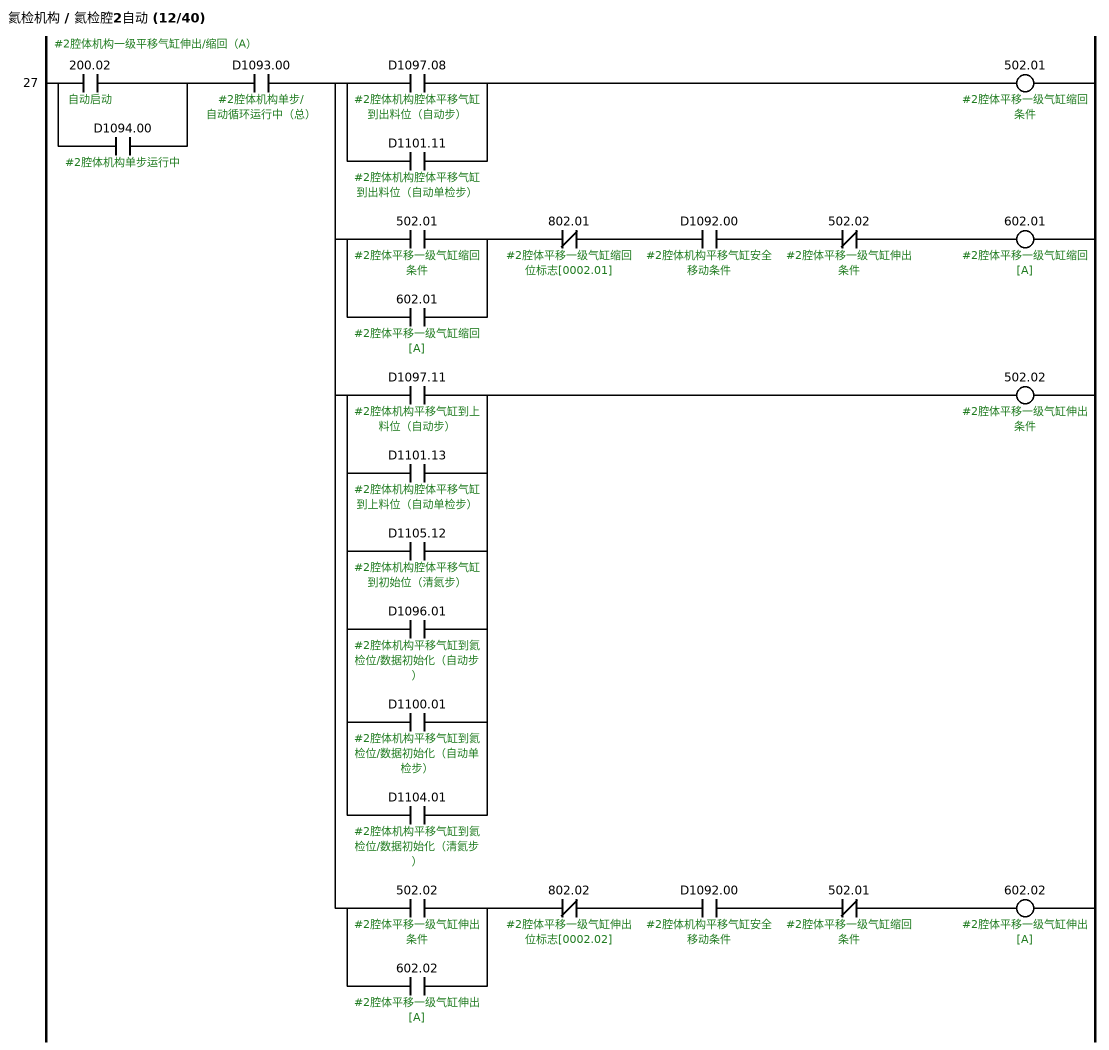
; [picture p264: 氦检机构 / 氦检腔2自动, rungs 27-27]
; rung 27: #2腔体机构一级平移气缸伸出/缩回（A）
LD 200.02  ; 自动启动
OR D1094.00  ; #2腔体机构单步运行中
AND D1093.00  ; #2腔体机构单步/自动循环运行中（总）
OUT TR0
LD D1097.08  ; #2腔体机构腔体平移气缸到出料位（自动步）
OR D1101.11  ; #2腔体机构腔体平移气缸到出料位（自动单检步）
ANDLD
OUT 502.01  ; #2腔体平移一级气缸缩回条件
LD TR0
LD 502.01  ; #2腔体平移一级气缸缩回条件
OR 602.01  ; #2腔体平移一级气缸缩回[A]
ANDLD
ANDNOT 802.01  ; #2腔体平移一级气缸缩回位标志[0002.01]
AND D1092.00  ; #2腔体机构平移气缸安全移动条件
ANDNOT 502.02  ; #2腔体平移一级气缸伸出条件
OUT 602.01  ; #2腔体平移一级气缸缩回[A]
LD TR0
LD D1097.11  ; #2腔体机构平移气缸到上料位（自动步）
OR D1101.13  ; #2腔体机构腔体平移气缸到上料位（自动单检步）
OR D1105.12  ; #2腔体机构腔体平移气缸到初始位（清氦步）
OR D1096.01  ; #2腔体机构平移气缸到氦检位/数据初始化（自动步）
OR D1100.01  ; #2腔体机构平移气缸到氦检位/数据初始化（自动单检步）
OR D1104.01  ; #2腔体机构平移气缸到氦检位/数据初始化（清氦步）
ANDLD
OUT 502.02  ; #2腔体平移一级气缸伸出条件
LD TR0
LD 502.02  ; #2腔体平移一级气缸伸出条件
OR 602.02  ; #2腔体平移一级气缸伸出[A]
ANDLD
ANDNOT 802.02  ; #2腔体平移一级气缸伸出位标志[0002.02]
AND D1092.00  ; #2腔体机构平移气缸安全移动条件
ANDNOT 502.01  ; #2腔体平移一级气缸缩回条件
OUT 602.02  ; #2腔体平移一级气缸伸出[A]

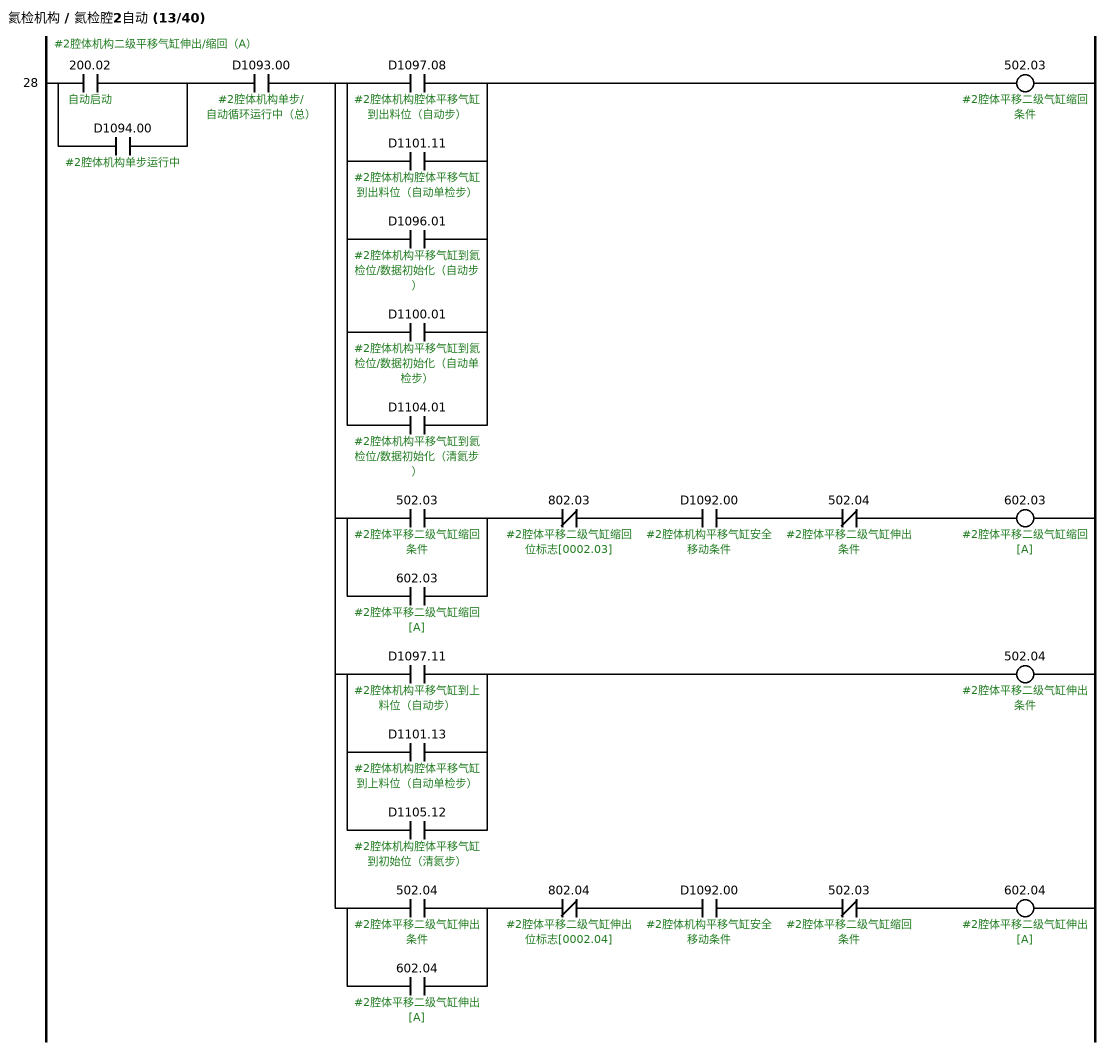
; rung 28: #2腔体机构二级平移气缸伸出/缩回（A）
LD 200.02  ; 自动启动
OR D1094.00  ; #2腔体机构单步运行中
AND D1093.00  ; #2腔体机构单步/自动循环运行中（总）
OUT TR0
LD D1097.08  ; #2腔体机构腔体平移气缸到出料位（自动步）
OR D1101.11  ; #2腔体机构腔体平移气缸到出料位（自动单检步）
OR D1096.01  ; #2腔体机构平移气缸到氦检位/数据初始化（自动步）
OR D1100.01  ; #2腔体机构平移气缸到氦检位/数据初始化（自动单检步）
OR D1104.01  ; #2腔体机构平移气缸到氦检位/数据初始化（清氦步）
ANDLD
OUT 502.03  ; #2腔体平移二级气缸缩回条件
LD TR0
LD 502.03  ; #2腔体平移二级气缸缩回条件
OR 602.03  ; #2腔体平移二级气缸缩回[A]
ANDLD
ANDNOT 802.03  ; #2腔体平移二级气缸缩回位标志[0002.03]
AND D1092.00  ; #2腔体机构平移气缸安全移动条件
ANDNOT 502.04  ; #2腔体平移二级气缸伸出条件
OUT 602.03  ; #2腔体平移二级气缸缩回[A]
LD TR0
LD D1097.11  ; #2腔体机构平移气缸到上料位（自动步）
OR D1101.13  ; #2腔体机构腔体平移气缸到上料位（自动单检步）
OR D1105.12  ; #2腔体机构腔体平移气缸到初始位（清氦步）
ANDLD
OUT 502.04  ; #2腔体平移二级气缸伸出条件
LD TR0
LD 502.04  ; #2腔体平移二级气缸伸出条件
OR 602.04  ; #2腔体平移二级气缸伸出[A]
ANDLD
ANDNOT 802.04  ; #2腔体平移二级气缸伸出位标志[0002.04]
AND D1092.00  ; #2腔体机构平移气缸安全移动条件
ANDNOT 502.03  ; #2腔体平移二级气缸缩回条件
OUT 602.04  ; #2腔体平移二级气缸伸出[A]

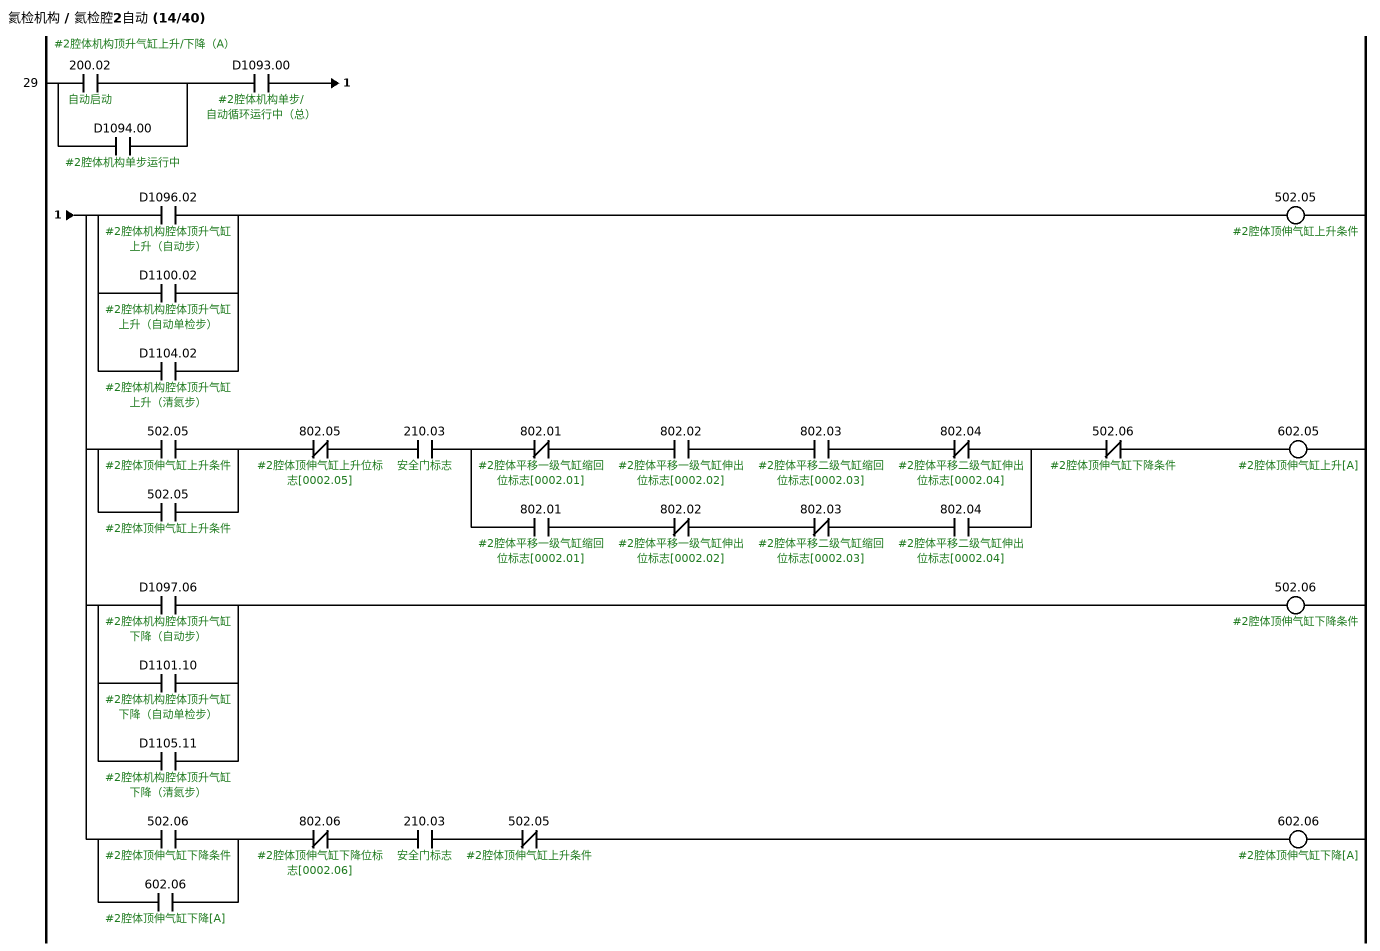
; rung 29: #2腔体机构顶升气缸上升/下降（A）
LD 200.02  ; 自动启动
OR D1094.00  ; #2腔体机构单步运行中
AND D1093.00  ; #2腔体机构单步/自动循环运行中（总）
OUT TR0
LD D1096.02  ; #2腔体机构腔体顶升气缸上升（自动步）
OR D1100.02  ; #2腔体机构腔体顶升气缸上升（自动单检步）
OR D1104.02  ; #2腔体机构腔体顶升气缸上升（清氦步）
ANDLD
OUT 502.05  ; #2腔体顶伸气缸上升条件
LD TR0
LD 502.05  ; #2腔体顶伸气缸上升条件
OR 502.05  ; #2腔体顶伸气缸上升条件
ANDLD
ANDNOT 802.05  ; #2腔体顶伸气缸上升位标志[0002.05]
AND 210.03  ; 安全门标志
LDNOT 802.01  ; #2腔体平移一级气缸缩回位标志[0002.01]
AND 802.02  ; #2腔体平移一级气缸伸出位标志[0002.02]
AND 802.03  ; #2腔体平移二级气缸缩回位标志[0002.03]
ANDNOT 802.04  ; #2腔体平移二级气缸伸出位标志[0002.04]
LD 802.01  ; #2腔体平移一级气缸缩回位标志[0002.01]
ANDNOT 802.02  ; #2腔体平移一级气缸伸出位标志[0002.02]
ANDNOT 802.03  ; #2腔体平移二级气缸缩回位标志[0002.03]
AND 802.04  ; #2腔体平移二级气缸伸出位标志[0002.04]
ORLD
ANDLD
ANDNOT 502.06  ; #2腔体顶伸气缸下降条件
OUT 602.05  ; #2腔体顶伸气缸上升[A]
LD TR0
LD D1097.06  ; #2腔体机构腔体顶升气缸下降（自动步）
OR D1101.10  ; #2腔体机构腔体顶升气缸下降（自动单检步）
OR D1105.11  ; #2腔体机构腔体顶升气缸下降（清氦步）
ANDLD
OUT 502.06  ; #2腔体顶伸气缸下降条件
LD TR0
LD 502.06  ; #2腔体顶伸气缸下降条件
OR 602.06  ; #2腔体顶伸气缸下降[A]
ANDLD
ANDNOT 802.06  ; #2腔体顶伸气缸下降位标志[0002.06]
AND 210.03  ; 安全门标志
ANDNOT 502.05  ; #2腔体顶伸气缸上升条件
OUT 602.06  ; #2腔体顶伸气缸下降[A]

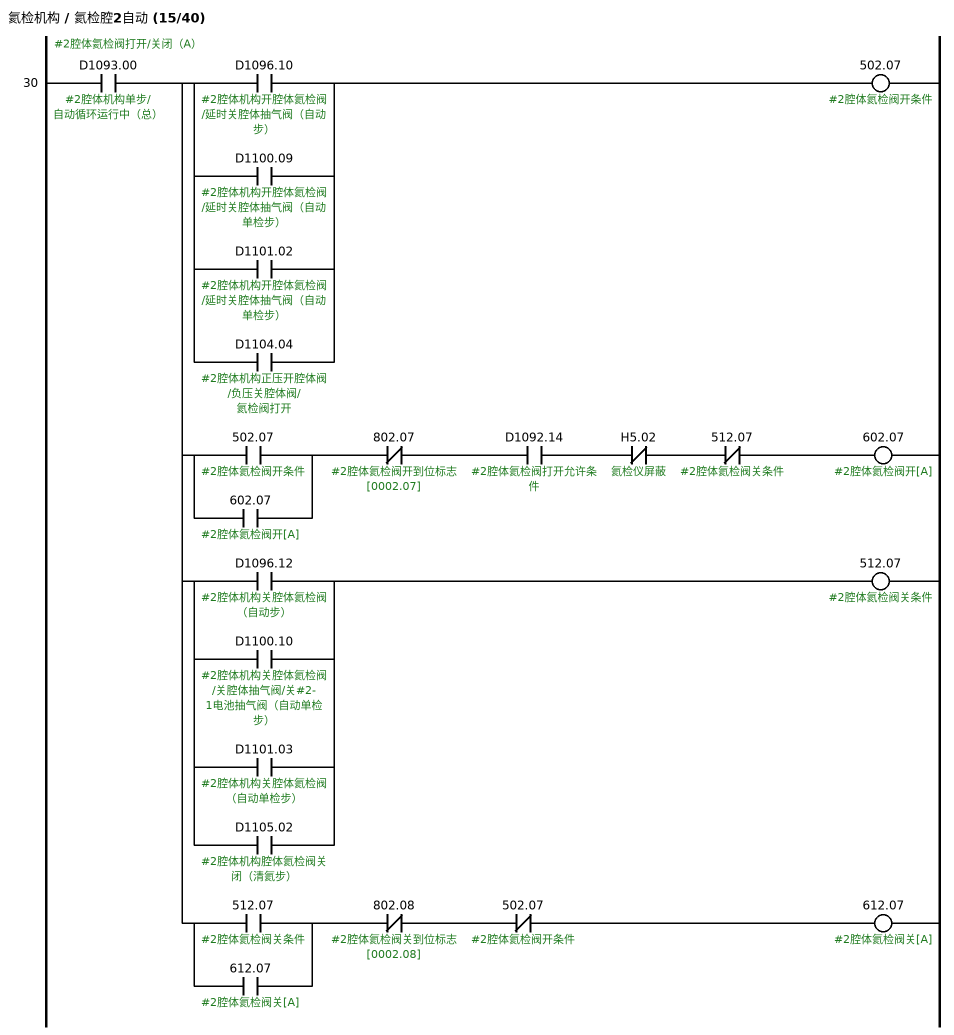
; rung 30: #2腔体氦检阀打开/关闭（A）
LD D1093.00  ; #2腔体机构单步/自动循环运行中（总）
OUT TR0
LD D1096.10  ; #2腔体机构开腔体氦检阀/延时关腔体抽气阀（自动步）
OR D1100.09  ; #2腔体机构开腔体氦检阀/延时关腔体抽气阀（自动单检步）
OR D1101.02  ; #2腔体机构开腔体氦检阀/延时关腔体抽气阀（自动单检步）
OR D1104.04  ; #2腔体机构正压开腔体阀/负压关腔体阀/氦检阀打开
ANDLD
OUT 502.07  ; #2腔体氦检阀开条件
LD TR0
LD 502.07  ; #2腔体氦检阀开条件
OR 602.07  ; #2腔体氦检阀开[A]
ANDLD
ANDNOT 802.07  ; #2腔体氦检阀开到位标志[0002.07]
AND D1092.14  ; #2腔体氦检阀打开允许条件
ANDNOT H5.02  ; 氦检仪屏蔽
ANDNOT 512.07  ; #2腔体氦检阀关条件
OUT 602.07  ; #2腔体氦检阀开[A]
LD TR0
LD D1096.12  ; #2腔体机构关腔体氦检阀（自动步）
OR D1100.10  ; #2腔体机构关腔体氦检阀/关腔体抽气阀/关#2-1电池抽气阀（自动单检步）
OR D1101.03  ; #2腔体机构关腔体氦检阀（自动单检步）
OR D1105.02  ; #2腔体机构腔体氦检阀关闭（清氦步）
ANDLD
OUT 512.07  ; #2腔体氦检阀关条件
LD TR0
LD 512.07  ; #2腔体氦检阀关条件
OR 612.07  ; #2腔体氦检阀关[A]
ANDLD
ANDNOT 802.08  ; #2腔体氦检阀关到位标志[0002.08]
ANDNOT 502.07  ; #2腔体氦检阀开条件
OUT 612.07  ; #2腔体氦检阀关[A]

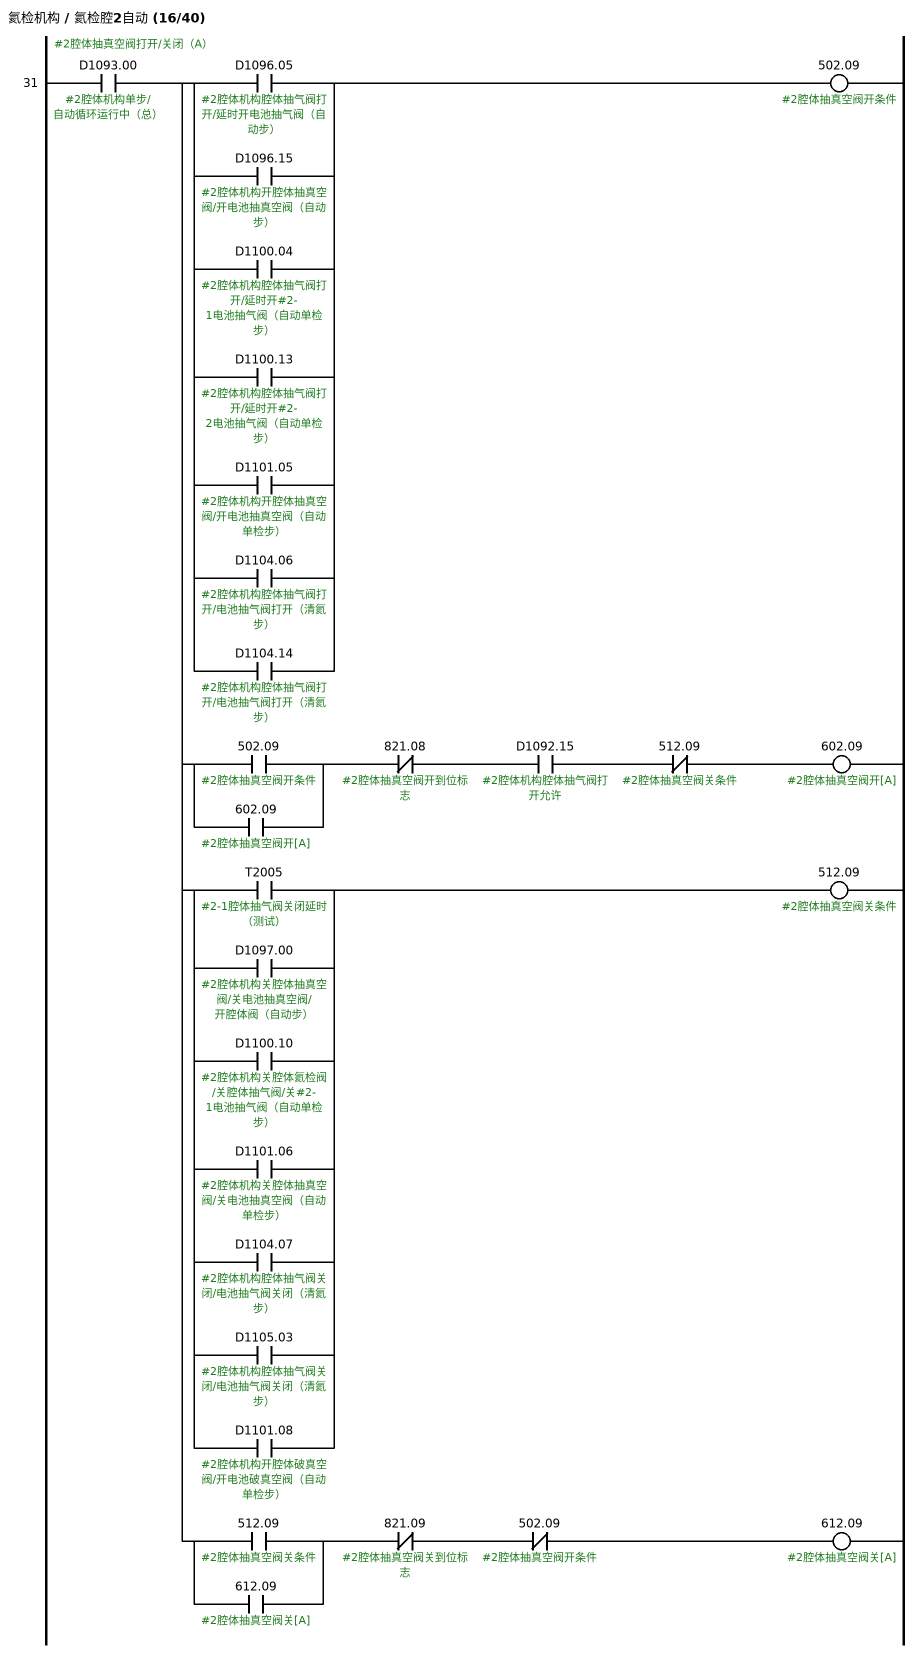
; rung 31: #2腔体抽真空阀打开/关闭（A）
LD D1093.00  ; #2腔体机构单步/自动循环运行中（总）
OUT TR0
LD D1096.05  ; #2腔体机构腔体抽气阀打开/延时开电池抽气阀（自动步）
OR D1096.15  ; #2腔体机构开腔体抽真空阀/开电池抽真空阀（自动步）
OR D1100.04  ; #2腔体机构腔体抽气阀打开/延时开#2-1电池抽气阀（自动单检步）
OR D1100.13  ; #2腔体机构腔体抽气阀打开/延时开#2-2电池抽气阀（自动单检步）
OR D1101.05  ; #2腔体机构开腔体抽真空阀/开电池抽真空阀（自动单检步）
OR D1104.06  ; #2腔体机构腔体抽气阀打开/电池抽气阀打开（清氦步）
OR D1104.14  ; #2腔体机构腔体抽气阀打开/电池抽气阀打开（清氦步）
ANDLD
OUT 502.09  ; #2腔体抽真空阀开条件
LD TR0
LD 502.09  ; #2腔体抽真空阀开条件
OR 602.09  ; #2腔体抽真空阀开[A]
ANDLD
ANDNOT 821.08  ; #2腔体抽真空阀开到位标志
AND D1092.15  ; #2腔体机构腔体抽气阀打开允许
ANDNOT 512.09  ; #2腔体抽真空阀关条件
OUT 602.09  ; #2腔体抽真空阀开[A]
LD TR0
LD T2005  ; #2-1腔体抽气阀关闭延时（测试）
OR D1097.00  ; #2腔体机构关腔体抽真空阀/关电池抽真空阀/开腔体阀（自动步）
OR D1100.10  ; #2腔体机构关腔体氦检阀/关腔体抽气阀/关#2-1电池抽气阀（自动单检步）
OR D1101.06  ; #2腔体机构关腔体抽真空阀/关电池抽真空阀（自动单检步）
OR D1104.07  ; #2腔体机构腔体抽气阀关闭/电池抽气阀关闭（清氦步）
OR D1105.03  ; #2腔体机构腔体抽气阀关闭/电池抽气阀关闭（清氦步）
OR D1101.08  ; #2腔体机构开腔体破真空阀/开电池破真空阀（自动单检步）
ANDLD
OUT 512.09  ; #2腔体抽真空阀关条件
LD TR0
LD 512.09  ; #2腔体抽真空阀关条件
OR 612.09  ; #2腔体抽真空阀关[A]
ANDLD
ANDNOT 821.09  ; #2腔体抽真空阀关到位标志
ANDNOT 502.09  ; #2腔体抽真空阀开条件
OUT 612.09  ; #2腔体抽真空阀关[A]

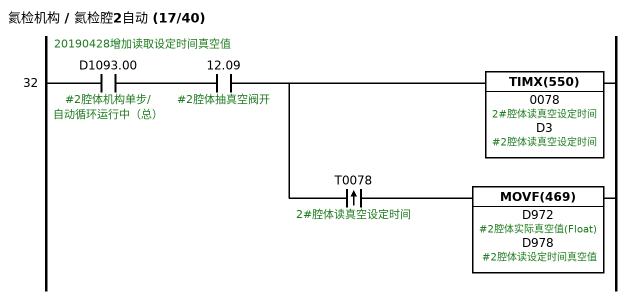
; rung 32: 20190428增加读取设定时间真空值
LD D1093.00  ; #2腔体机构单步/自动循环运行中（总）
AND 12.09  ; #2腔体抽真空阀开
TIMX(550) 0078 D3  ; #2腔体读真空设定时间, 2#腔体读真空设定时间
@AND T0078  ; 2#腔体读真空设定时间
MOVF(469) D972 D978  ; #2腔体实际真空值(Float), #2腔体读设定时间真空值

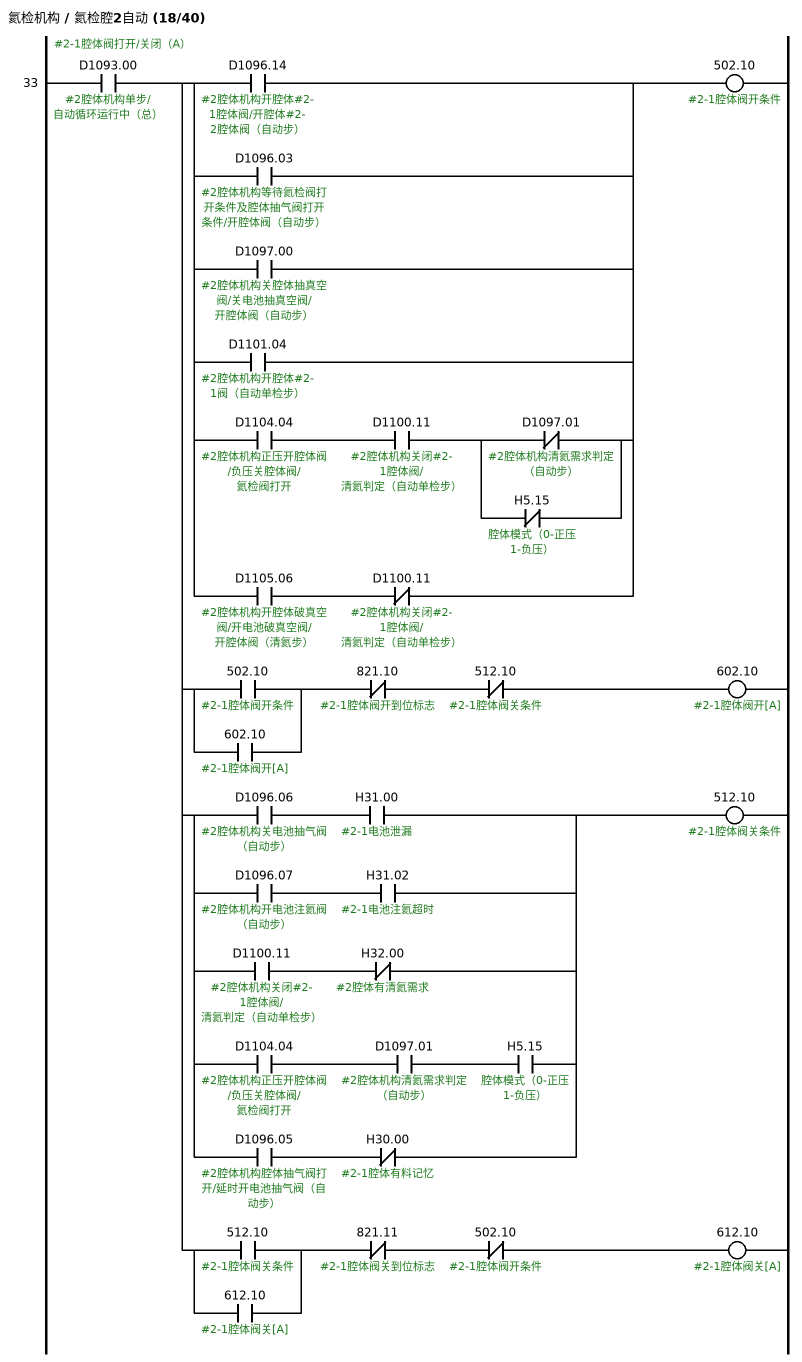
; rung 33: #2-1腔体阀打开/关闭（A）
LD D1093.00  ; #2腔体机构单步/自动循环运行中（总）
OUT TR0
LD D1096.14  ; #2腔体机构开腔体#2-1腔体阀/开腔体#2-2腔体阀（自动步）
OR D1096.03  ; #2腔体机构等待氦检阀打开条件及腔体抽气阀打开条件/开腔体阀（自动步）
OR D1097.00  ; #2腔体机构关腔体抽真空阀/关电池抽真空阀/开腔体阀（自动步）
OR D1101.04  ; #2腔体机构开腔体#2-1阀（自动单检步）
LD D1104.04  ; #2腔体机构正压开腔体阀/负压关腔体阀/氦检阀打开
AND D1100.11  ; #2腔体机构关闭#2-1腔体阀/清氦判定（自动单检步）
LDNOT D1097.01  ; #2腔体机构清氦需求判定（自动步）
ORNOT H5.15  ; 腔体模式（0-正压 1-负压）
ANDLD
ORLD
LD D1105.06  ; #2腔体机构开腔体破真空阀/开电池破真空阀/开腔体阀（清氦步）
ANDNOT D1100.11  ; #2腔体机构关闭#2-1腔体阀/清氦判定（自动单检步）
ORLD
ANDLD
OUT 502.10  ; #2-1腔体阀开条件
LD TR0
LD 502.10  ; #2-1腔体阀开条件
OR 602.10  ; #2-1腔体阀开[A]
ANDLD
ANDNOT 821.10  ; #2-1腔体阀开到位标志
ANDNOT 512.10  ; #2-1腔体阀关条件
OUT 602.10  ; #2-1腔体阀开[A]
LD TR0
LD D1096.06  ; #2腔体机构关电池抽气阀（自动步）
AND H31.00  ; #2-1电池泄漏
LD D1096.07  ; #2腔体机构开电池注氦阀（自动步）
AND H31.02  ; #2-1电池注氦超时
ORLD
LD D1100.11  ; #2腔体机构关闭#2-1腔体阀/清氦判定（自动单检步）
ANDNOT H32.00  ; #2腔体有清氦需求
ORLD
LD D1104.04  ; #2腔体机构正压开腔体阀/负压关腔体阀/氦检阀打开
AND D1097.01  ; #2腔体机构清氦需求判定（自动步）
AND H5.15  ; 腔体模式（0-正压 1-负压）
ORLD
LD D1096.05  ; #2腔体机构腔体抽气阀打开/延时开电池抽气阀（自动步）  // #1-1无料时不测试
ANDNOT H30.00  ; #2-1腔体有料记忆
ORLD
ANDLD
OUT 512.10  ; #2-1腔体阀关条件
LD TR0
LD 512.10  ; #2-1腔体阀关条件
OR 612.10  ; #2-1腔体阀关[A]
ANDLD
ANDNOT 821.11  ; #2-1腔体阀关到位标志
ANDNOT 502.10  ; #2-1腔体阀开条件
OUT 612.10  ; #2-1腔体阀关[A]

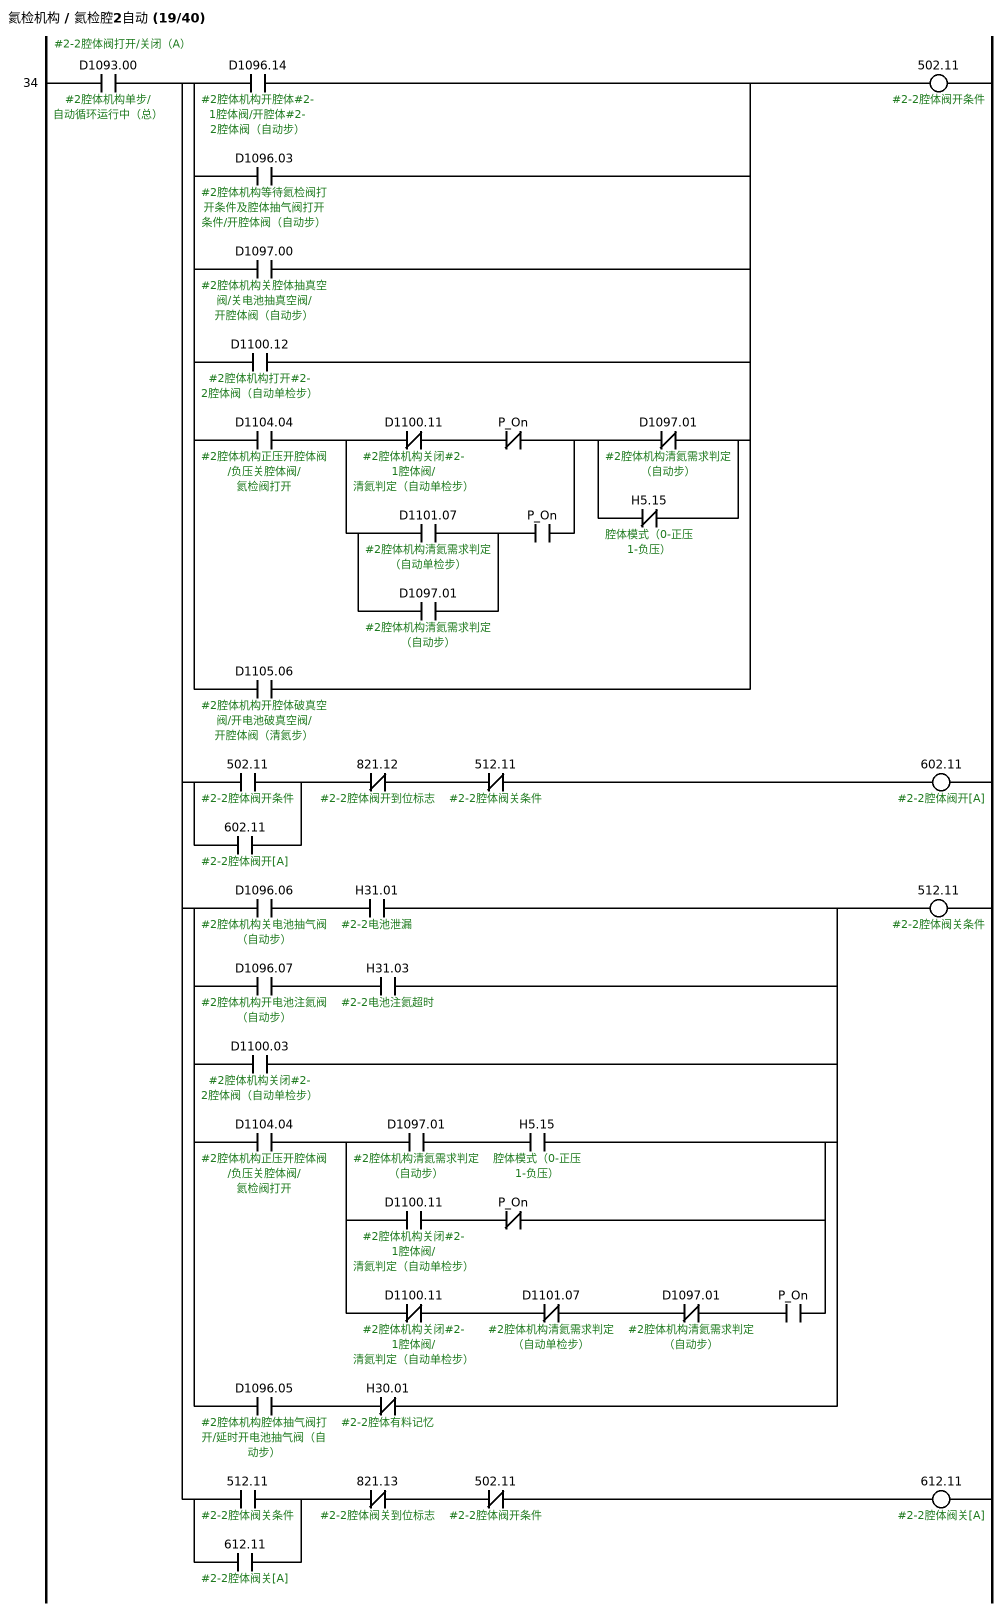
; rung 34: #2-2腔体阀打开/关闭（A）
LD D1093.00  ; #2腔体机构单步/自动循环运行中（总）
OUT TR0
LD D1096.14  ; #2腔体机构开腔体#2-1腔体阀/开腔体#2-2腔体阀（自动步）
OR D1096.03  ; #2腔体机构等待氦检阀打开条件及腔体抽气阀打开条件/开腔体阀（自动步）
OR D1097.00  ; #2腔体机构关腔体抽真空阀/关电池抽真空阀/开腔体阀（自动步）
OR D1100.12  ; #2腔体机构打开#2-2腔体阀（自动单检步）
LD D1104.04  ; #2腔体机构正压开腔体阀/负压关腔体阀/氦检阀打开
LDNOT D1100.11  ; #2腔体机构关闭#2-1腔体阀/清氦判定（自动单检步）
ANDNOT P_On
LD D1101.07  ; #2腔体机构清氦需求判定（自动单检步）
OR D1097.01  ; #2腔体机构清氦需求判定（自动步）
AND P_On
ORLD
ANDLD
LDNOT D1097.01  ; #2腔体机构清氦需求判定（自动步）
ORNOT H5.15  ; 腔体模式（0-正压 1-负压）
ANDLD
ORLD
OR D1105.06  ; #2腔体机构开腔体破真空阀/开电池破真空阀/开腔体阀（清氦步）
ANDLD
OUT 502.11  ; #2-2腔体阀开条件
LD TR0
LD 502.11  ; #2-2腔体阀开条件
OR 602.11  ; #2-2腔体阀开[A]
ANDLD
ANDNOT 821.12  ; #2-2腔体阀开到位标志
ANDNOT 512.11  ; #2-2腔体阀关条件
OUT 602.11  ; #2-2腔体阀开[A]
LD TR0
LD D1096.06  ; #2腔体机构关电池抽气阀（自动步）
AND H31.01  ; #2-2电池泄漏
LD D1096.07  ; #2腔体机构开电池注氦阀（自动步）
AND H31.03  ; #2-2电池注氦超时
ORLD
OR D1100.03  ; #2腔体机构关闭#2-2腔体阀（自动单检步）
LD D1104.04  ; #2腔体机构正压开腔体阀/负压关腔体阀/氦检阀打开
LD D1097.01  ; #2腔体机构清氦需求判定（自动步）
AND H5.15  ; 腔体模式（0-正压 1-负压）
LD D1100.11  ; #2腔体机构关闭#2-1腔体阀/清氦判定（自动单检步）
ANDNOT P_On
ORLD
LDNOT D1100.11  ; #2腔体机构关闭#2-1腔体阀/清氦判定（自动单检步）
ANDNOT D1101.07  ; #2腔体机构清氦需求判定（自动单检步）
ANDNOT D1097.01  ; #2腔体机构清氦需求判定（自动步）
AND P_On
ORLD
ANDLD
ORLD
LD D1096.05  ; #2腔体机构腔体抽气阀打开/延时开电池抽气阀（自动步）  // #1-2无料时不测试
ANDNOT H30.01  ; #2-2腔体有料记忆
ORLD
ANDLD
OUT 512.11  ; #2-2腔体阀关条件
LD TR0
LD 512.11  ; #2-2腔体阀关条件
OR 612.11  ; #2-2腔体阀关[A]
ANDLD
ANDNOT 821.13  ; #2-2腔体阀关到位标志
ANDNOT 502.11  ; #2-2腔体阀开条件
OUT 612.11  ; #2-2腔体阀关[A]

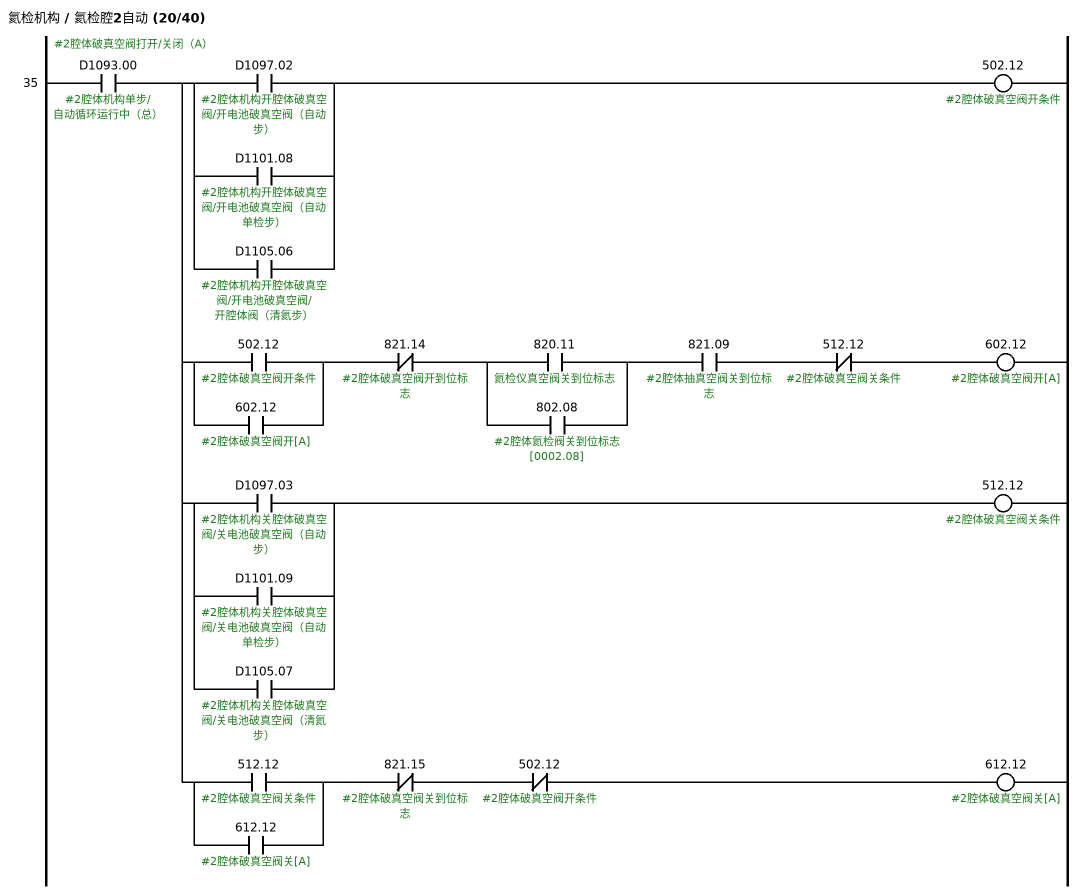
; rung 35: #2腔体破真空阀打开/关闭（A）
LD D1093.00  ; #2腔体机构单步/自动循环运行中（总）
OUT TR0
LD D1097.02  ; #2腔体机构开腔体破真空阀/开电池破真空阀（自动步）
OR D1101.08  ; #2腔体机构开腔体破真空阀/开电池破真空阀（自动单检步）
OR D1105.06  ; #2腔体机构开腔体破真空阀/开电池破真空阀/开腔体阀（清氦步）
ANDLD
OUT 502.12  ; #2腔体破真空阀开条件
LD TR0
LD 502.12  ; #2腔体破真空阀开条件
OR 602.12  ; #2腔体破真空阀开[A]
ANDLD
ANDNOT 821.14  ; #2腔体破真空阀开到位标志
LD 820.11  ; 氦检仪真空阀关到位标志
OR 802.08  ; #2腔体氦检阀关到位标志[0002.08]
ANDLD
AND 821.09  ; #2腔体抽真空阀关到位标志
ANDNOT 512.12  ; #2腔体破真空阀关条件
OUT 602.12  ; #2腔体破真空阀开[A]
LD TR0
LD D1097.03  ; #2腔体机构关腔体破真空阀/关电池破真空阀（自动步）
OR D1101.09  ; #2腔体机构关腔体破真空阀/关电池破真空阀（自动单检步）
OR D1105.07  ; #2腔体机构关腔体破真空阀/关电池破真空阀（清氦步）
ANDLD
OUT 512.12  ; #2腔体破真空阀关条件
LD TR0
LD 512.12  ; #2腔体破真空阀关条件
OR 612.12  ; #2腔体破真空阀关[A]
ANDLD
ANDNOT 821.15  ; #2腔体破真空阀关到位标志
ANDNOT 502.12  ; #2腔体破真空阀开条件
OUT 612.12  ; #2腔体破真空阀关[A]

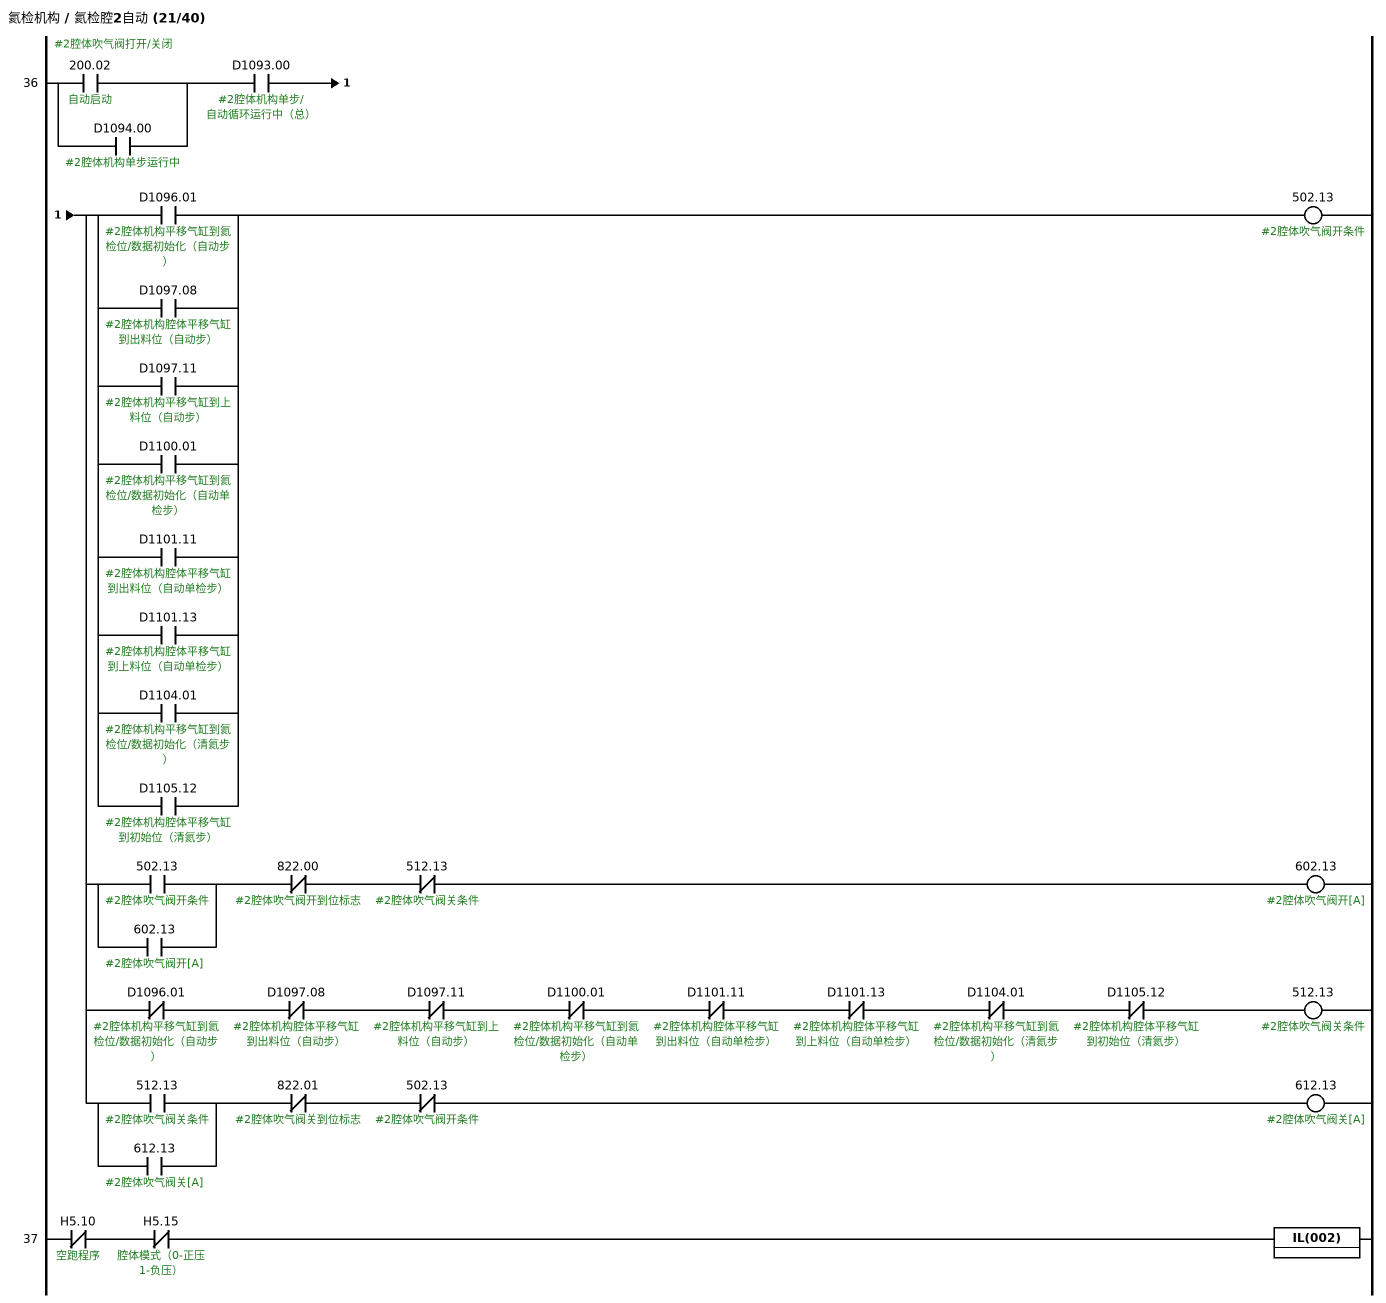
; rung 36: #2腔体吹气阀打开/关闭
LD 200.02  ; 自动启动
OR D1094.00  ; #2腔体机构单步运行中
AND D1093.00  ; #2腔体机构单步/自动循环运行中（总）
OUT TR0
LD D1096.01  ; #2腔体机构平移气缸到氦检位/数据初始化（自动步）
OR D1097.08  ; #2腔体机构腔体平移气缸到出料位（自动步）
OR D1097.11  ; #2腔体机构平移气缸到上料位（自动步）
OR D1100.01  ; #2腔体机构平移气缸到氦检位/数据初始化（自动单检步）
OR D1101.11  ; #2腔体机构腔体平移气缸到出料位（自动单检步）
OR D1101.13  ; #2腔体机构腔体平移气缸到上料位（自动单检步）
OR D1104.01  ; #2腔体机构平移气缸到氦检位/数据初始化（清氦步）
OR D1105.12  ; #2腔体机构腔体平移气缸到初始位（清氦步）
ANDLD
OUT 502.13  ; #2腔体吹气阀开条件
LD TR0
LD 502.13  ; #2腔体吹气阀开条件
OR 602.13  ; #2腔体吹气阀开[A]
ANDLD
ANDNOT 822.00  ; #2腔体吹气阀开到位标志
ANDNOT 512.13  ; #2腔体吹气阀关条件
OUT 602.13  ; #2腔体吹气阀开[A]
LD TR0
ANDNOT D1096.01  ; #2腔体机构平移气缸到氦检位/数据初始化（自动步）
ANDNOT D1097.08  ; #2腔体机构腔体平移气缸到出料位（自动步）
ANDNOT D1097.11  ; #2腔体机构平移气缸到上料位（自动步）
ANDNOT D1100.01  ; #2腔体机构平移气缸到氦检位/数据初始化（自动单检步）
ANDNOT D1101.11  ; #2腔体机构腔体平移气缸到出料位（自动单检步）
ANDNOT D1101.13  ; #2腔体机构腔体平移气缸到上料位（自动单检步）
ANDNOT D1104.01  ; #2腔体机构平移气缸到氦检位/数据初始化（清氦步）
ANDNOT D1105.12  ; #2腔体机构腔体平移气缸到初始位（清氦步）
OUT 512.13  ; #2腔体吹气阀关条件
LD TR0
LD 512.13  ; #2腔体吹气阀关条件
OR 612.13  ; #2腔体吹气阀关[A]
ANDLD
ANDNOT 822.01  ; #2腔体吹气阀关到位标志
ANDNOT 502.13  ; #2腔体吹气阀开条件
OUT 612.13  ; #2腔体吹气阀关[A]
; rung 37
LDNOT H5.10  ; 空跑程序
ANDNOT H5.15  ; 腔体模式（0-正压 1-负压）
IL(002)

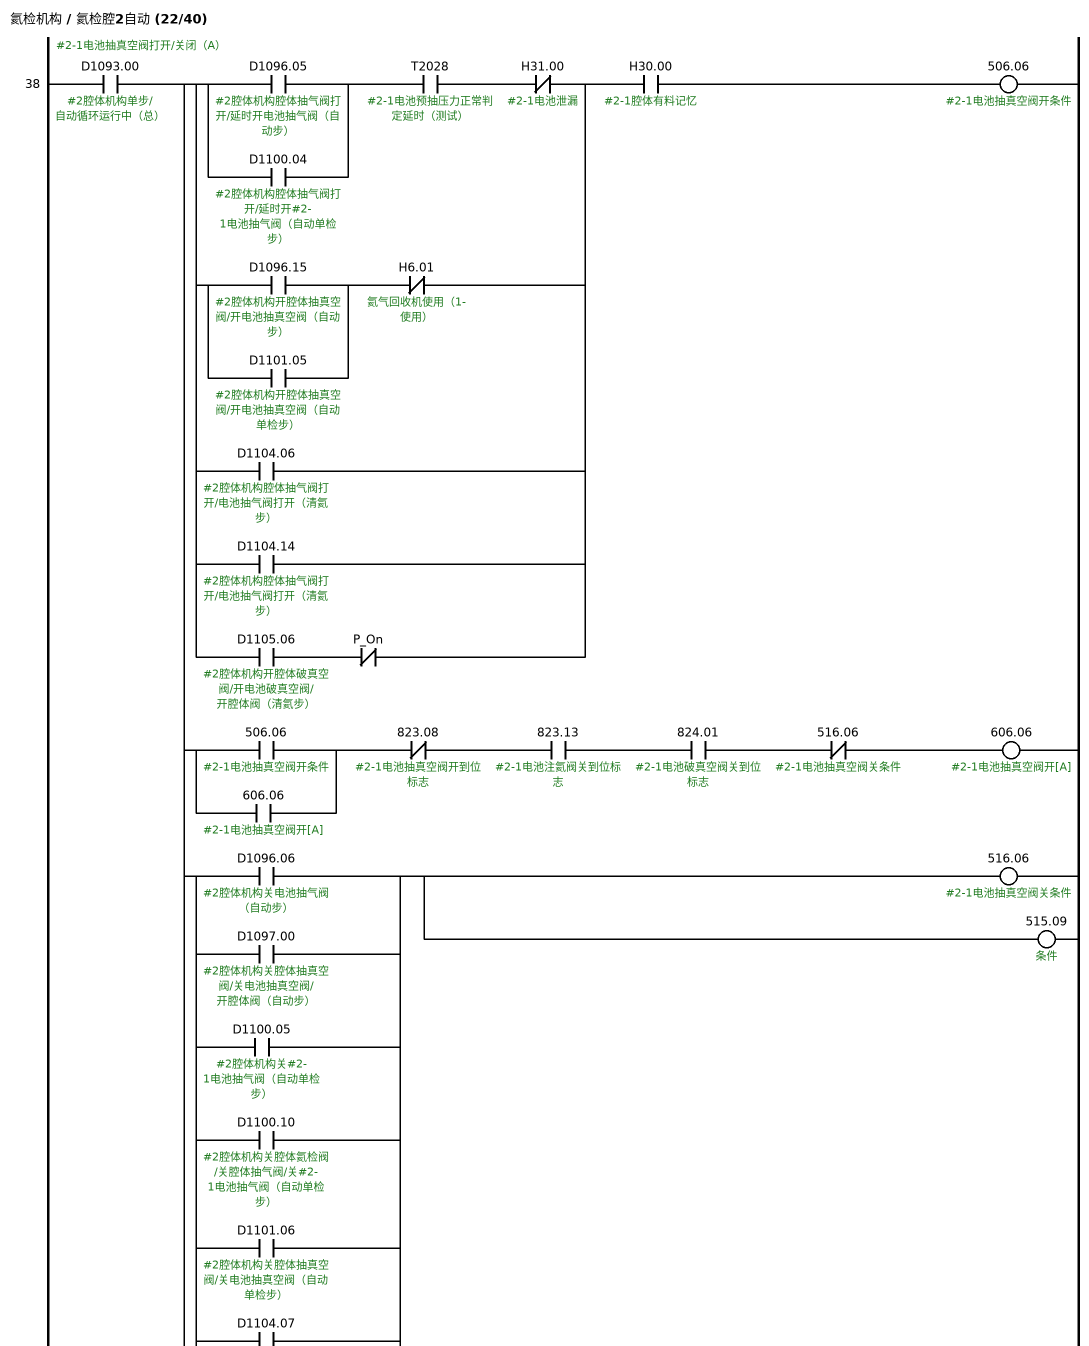

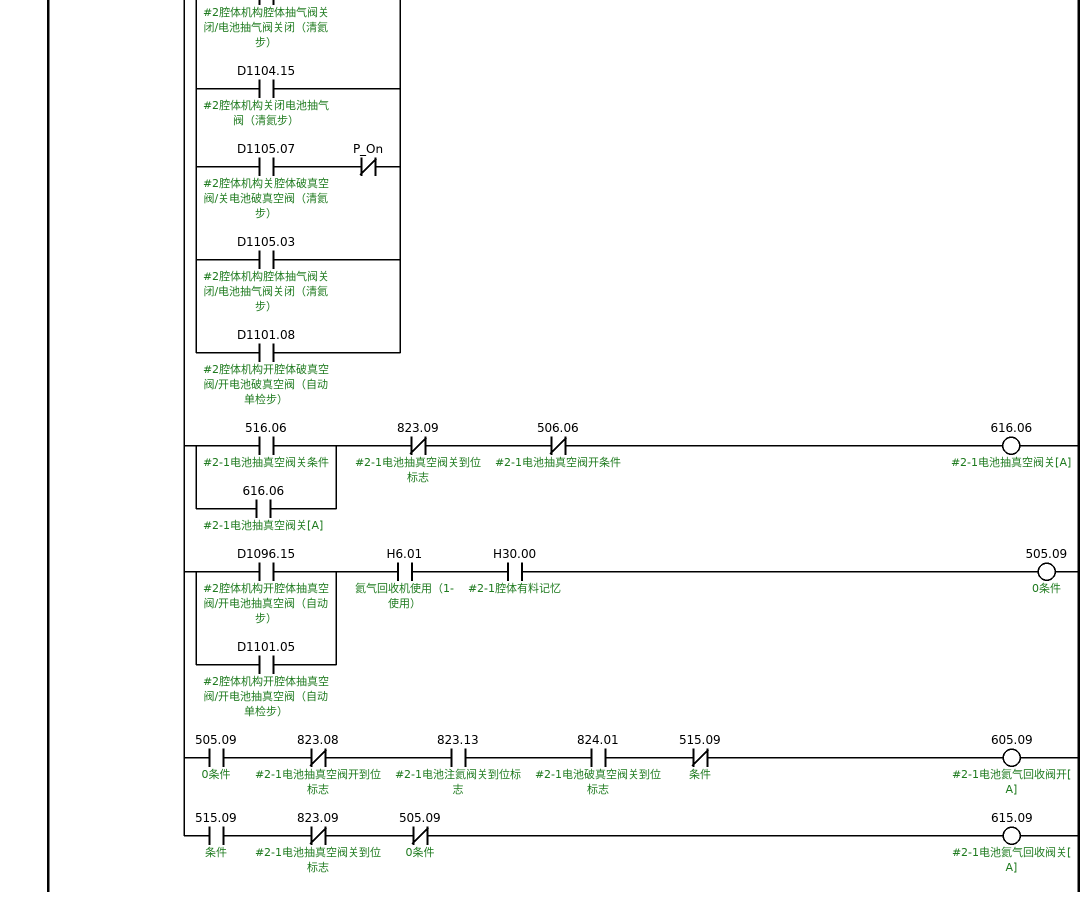
; rung 38: #2-1电池抽真空阀打开/关闭（A）
LD D1093.00  ; #2腔体机构单步/自动循环运行中（总）
OUT TR0
LD D1096.05  ; #2腔体机构腔体抽气阀打开/延时开电池抽气阀（自动步）
OR D1100.04  ; #2腔体机构腔体抽气阀打开/延时开#2-1电池抽气阀（自动单检步）
AND T2028  ; #2-1电池预抽压力正常判定延时（测试）
ANDNOT H31.00  ; #2-1电池泄漏
LD D1096.15  ; #2腔体机构开腔体抽真空阀/开电池抽真空阀（自动步）
OR D1101.05  ; #2腔体机构开腔体抽真空阀/开电池抽真空阀（自动单检步）
ANDNOT H6.01  ; 氦气回收机使用（1-使用）
ORLD
OR D1104.06  ; #2腔体机构腔体抽气阀打开/电池抽气阀打开（清氦步）
OR D1104.14  ; #2腔体机构腔体抽气阀打开/电池抽气阀打开（清氦步）
LD D1105.06  ; #2腔体机构开腔体破真空阀/开电池破真空阀/开腔体阀（清氦步）
ANDNOT P_On
ORLD
ANDLD
AND H30.00  ; #2-1腔体有料记忆
OUT 506.06  ; #2-1电池抽真空阀开条件
LD TR0
LD 506.06  ; #2-1电池抽真空阀开条件
OR 606.06  ; #2-1电池抽真空阀开[A]
ANDLD
ANDNOT 823.08  ; #2-1电池抽真空阀开到位标志
AND 823.13  ; #2-1电池注氦阀关到位标志
AND 824.01  ; #2-1电池破真空阀关到位标志
ANDNOT 516.06  ; #2-1电池抽真空阀关条件
OUT 606.06  ; #2-1电池抽真空阀开[A]
LD TR0
LD D1096.06  ; #2腔体机构关电池抽气阀（自动步）
OR D1097.00  ; #2腔体机构关腔体抽真空阀/关电池抽真空阀/开腔体阀（自动步）
OR D1100.05  ; #2腔体机构关#2-1电池抽气阀（自动单检步）
OR D1100.10  ; #2腔体机构关腔体氦检阀/关腔体抽气阀/关#2-1电池抽气阀（自动单检步）
OR D1101.06  ; #2腔体机构关腔体抽真空阀/关电池抽真空阀（自动单检步）
OR D1104.07  ; #2腔体机构腔体抽气阀关闭/电池抽气阀关闭（清氦步）
OR D1104.15  ; #2腔体机构关闭电池抽气阀（清氦步）
LD D1105.07  ; #2腔体机构关腔体破真空阀/关电池破真空阀（清氦步）
ANDNOT P_On
ORLD
OR D1105.03  ; #2腔体机构腔体抽气阀关闭/电池抽气阀关闭（清氦步）
OR D1101.08  ; #2腔体机构开腔体破真空阀/开电池破真空阀（自动单检步）
ANDLD
OUT 516.06  ; #2-1电池抽真空阀关条件
OUT 515.09  ; 条件
LD TR0
LD 516.06  ; #2-1电池抽真空阀关条件
OR 616.06  ; #2-1电池抽真空阀关[A]
ANDLD
ANDNOT 823.09  ; #2-1电池抽真空阀关到位标志
ANDNOT 506.06  ; #2-1电池抽真空阀开条件
OUT 616.06  ; #2-1电池抽真空阀关[A]
LD TR0
LD D1096.15  ; #2腔体机构开腔体抽真空阀/开电池抽真空阀（自动步）
OR D1101.05  ; #2腔体机构开腔体抽真空阀/开电池抽真空阀（自动单检步）
ANDLD
AND H6.01  ; 氦气回收机使用（1-使用）
AND H30.00  ; #2-1腔体有料记忆
OUT 505.09  ; 0条件
LD TR0
AND 505.09  ; 0条件
ANDNOT 823.08  ; #2-1电池抽真空阀开到位标志
AND 823.13  ; #2-1电池注氦阀关到位标志
AND 824.01  ; #2-1电池破真空阀关到位标志
ANDNOT 515.09  ; 条件
OUT 605.09  ; #2-1电池氦气回收阀开[A]
LD TR0
AND 515.09  ; 条件
ANDNOT 823.09  ; #2-1电池抽真空阀关到位标志
ANDNOT 505.09  ; 0条件
OUT 615.09  ; #2-1电池氦气回收阀关[A]

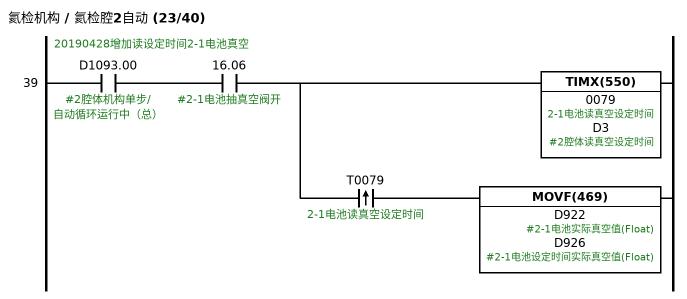
; rung 39: 20190428增加读设定时间2-1电池真空
LD D1093.00  ; #2腔体机构单步/自动循环运行中（总）
AND 16.06  ; #2-1电池抽真空阀开
TIMX(550) 0079 D3  ; #2腔体读真空设定时间, 2-1电池读真空设定时间
@AND T0079  ; 2-1电池读真空设定时间
MOVF(469) D922 D926  ; #2-1电池实际真空值(Float), #2-1电池设定时间实际真空值(Float)

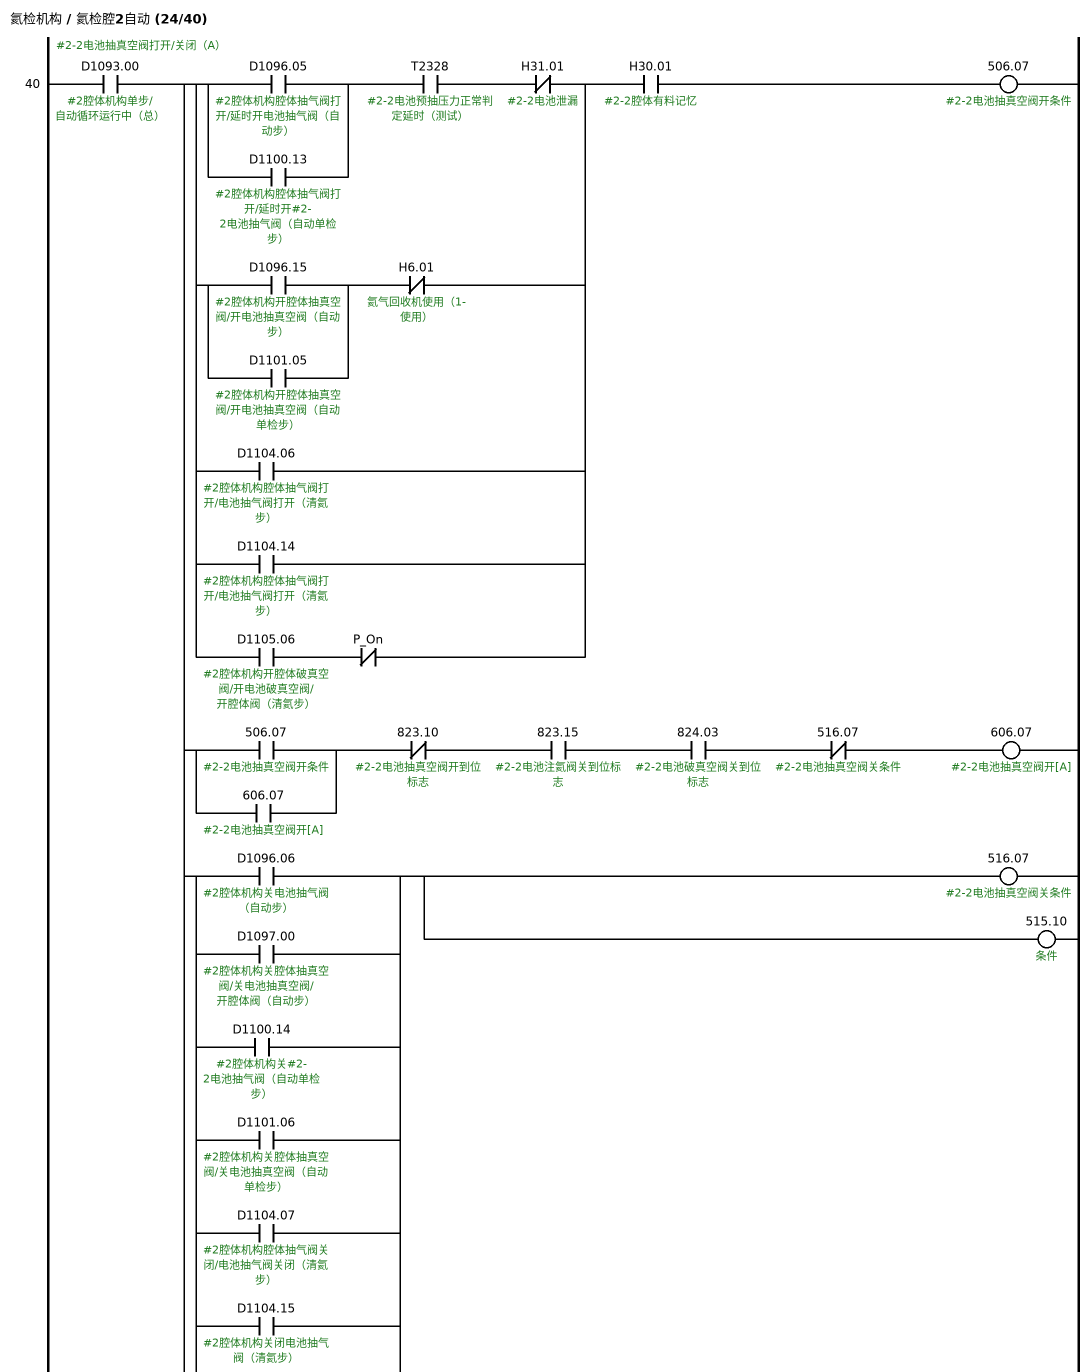

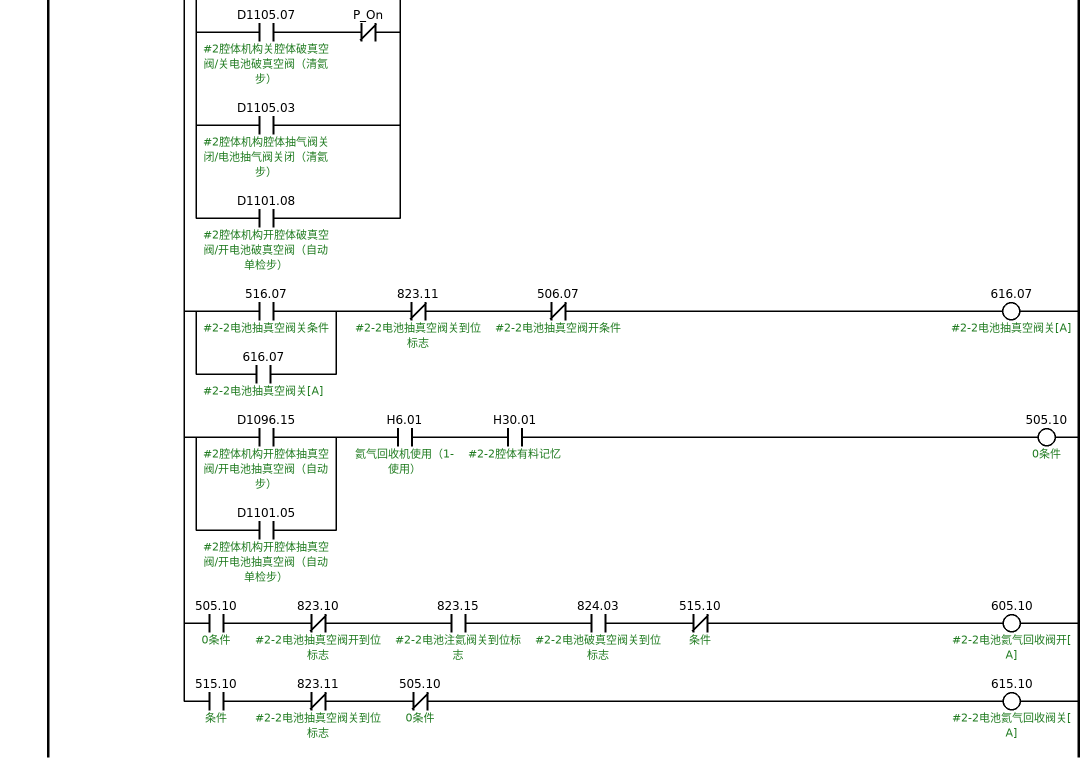
; rung 40: #2-2电池抽真空阀打开/关闭（A）
LD D1093.00  ; #2腔体机构单步/自动循环运行中（总）
OUT TR0
LD D1096.05  ; #2腔体机构腔体抽气阀打开/延时开电池抽气阀（自动步）
OR D1100.13  ; #2腔体机构腔体抽气阀打开/延时开#2-2电池抽气阀（自动单检步）
AND T2328  ; #2-2电池预抽压力正常判定延时（测试）
ANDNOT H31.01  ; #2-2电池泄漏
LD D1096.15  ; #2腔体机构开腔体抽真空阀/开电池抽真空阀（自动步）
OR D1101.05  ; #2腔体机构开腔体抽真空阀/开电池抽真空阀（自动单检步）
ANDNOT H6.01  ; 氦气回收机使用（1-使用）
ORLD
OR D1104.06  ; #2腔体机构腔体抽气阀打开/电池抽气阀打开（清氦步）
OR D1104.14  ; #2腔体机构腔体抽气阀打开/电池抽气阀打开（清氦步）
LD D1105.06  ; #2腔体机构开腔体破真空阀/开电池破真空阀/开腔体阀（清氦步）
ANDNOT P_On
ORLD
ANDLD
AND H30.01  ; #2-2腔体有料记忆
OUT 506.07  ; #2-2电池抽真空阀开条件
LD TR0
LD 506.07  ; #2-2电池抽真空阀开条件
OR 606.07  ; #2-2电池抽真空阀开[A]
ANDLD
ANDNOT 823.10  ; #2-2电池抽真空阀开到位标志
AND 823.15  ; #2-2电池注氦阀关到位标志
AND 824.03  ; #2-2电池破真空阀关到位标志
ANDNOT 516.07  ; #2-2电池抽真空阀关条件
OUT 606.07  ; #2-2电池抽真空阀开[A]
LD TR0
LD D1096.06  ; #2腔体机构关电池抽气阀（自动步）
OR D1097.00  ; #2腔体机构关腔体抽真空阀/关电池抽真空阀/开腔体阀（自动步）
OR D1100.14  ; #2腔体机构关#2-2电池抽气阀（自动单检步）
OR D1101.06  ; #2腔体机构关腔体抽真空阀/关电池抽真空阀（自动单检步）
OR D1104.07  ; #2腔体机构腔体抽气阀关闭/电池抽气阀关闭（清氦步）
OR D1104.15  ; #2腔体机构关闭电池抽气阀（清氦步）
LD D1105.07  ; #2腔体机构关腔体破真空阀/关电池破真空阀（清氦步）
ANDNOT P_On
ORLD
OR D1105.03  ; #2腔体机构腔体抽气阀关闭/电池抽气阀关闭（清氦步）
OR D1101.08  ; #2腔体机构开腔体破真空阀/开电池破真空阀（自动单检步）
ANDLD
OUT 516.07  ; #2-2电池抽真空阀关条件
OUT 515.10  ; 条件
LD TR0
LD 516.07  ; #2-2电池抽真空阀关条件
OR 616.07  ; #2-2电池抽真空阀关[A]
ANDLD
ANDNOT 823.11  ; #2-2电池抽真空阀关到位标志
ANDNOT 506.07  ; #2-2电池抽真空阀开条件
OUT 616.07  ; #2-2电池抽真空阀关[A]
LD TR0
LD D1096.15  ; #2腔体机构开腔体抽真空阀/开电池抽真空阀（自动步）
OR D1101.05  ; #2腔体机构开腔体抽真空阀/开电池抽真空阀（自动单检步）
ANDLD
AND H6.01  ; 氦气回收机使用（1-使用）
AND H30.01  ; #2-2腔体有料记忆
OUT 505.10  ; 0条件
LD TR0
AND 505.10  ; 0条件
ANDNOT 823.10  ; #2-2电池抽真空阀开到位标志
AND 823.15  ; #2-2电池注氦阀关到位标志
AND 824.03  ; #2-2电池破真空阀关到位标志
ANDNOT 515.10  ; 条件
OUT 605.10  ; #2-2电池氦气回收阀开[A]
LD TR0
AND 515.10  ; 条件
ANDNOT 823.11  ; #2-2电池抽真空阀关到位标志
ANDNOT 505.10  ; 0条件
OUT 615.10  ; #2-2电池氦气回收阀关[A]

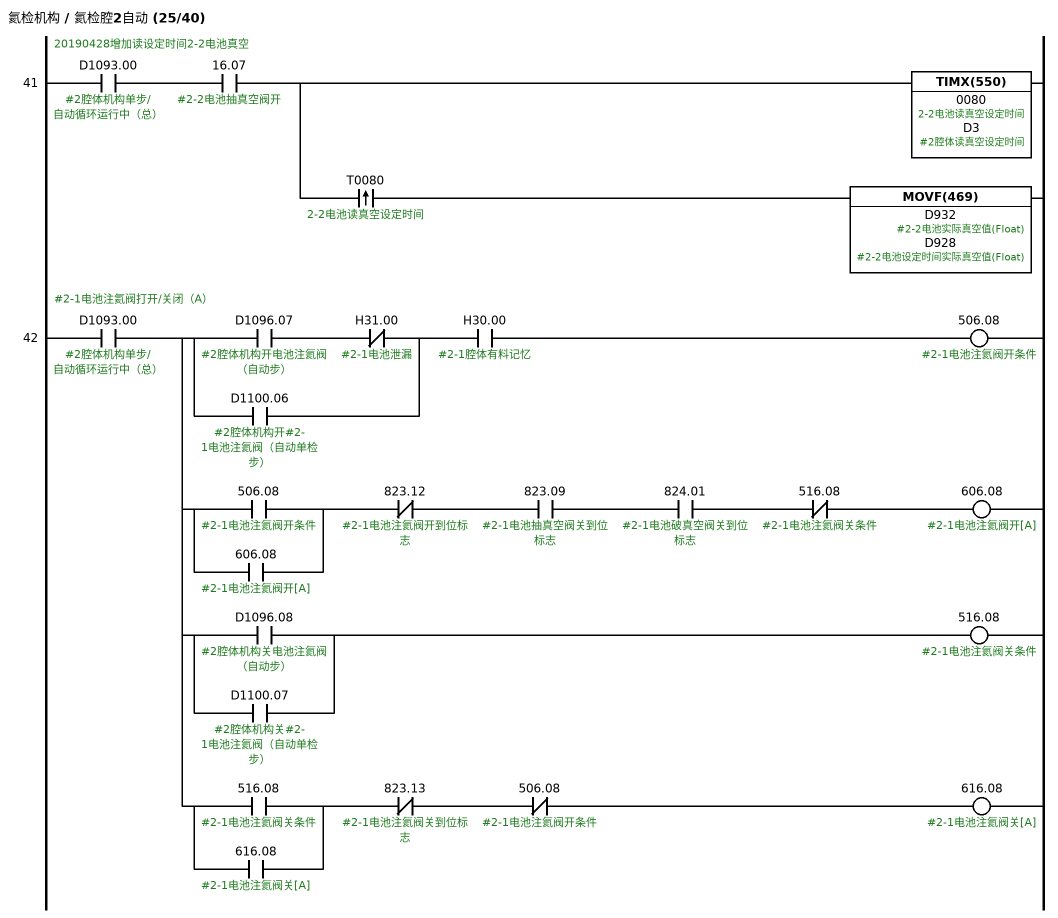
; rung 41: 20190428增加读设定时间2-2电池真空
LD D1093.00  ; #2腔体机构单步/自动循环运行中（总）
AND 16.07  ; #2-2电池抽真空阀开
TIMX(550) 0080 D3  ; #2腔体读真空设定时间, 2-2电池读真空设定时间
@AND T0080  ; 2-2电池读真空设定时间
MOVF(469) D932 D928  ; #2-2电池实际真空值(Float), #2-2电池设定时间实际真空值(Float)
; rung 42: #2-1电池注氦阀打开/关闭（A）
LD D1093.00  ; #2腔体机构单步/自动循环运行中（总）
OUT TR0
LD D1096.07  ; #2腔体机构开电池注氦阀（自动步）
ANDNOT H31.00  ; #2-1电池泄漏
OR D1100.06  ; #2腔体机构开#2-1电池注氦阀（自动单检步）
ANDLD
AND H30.00  ; #2-1腔体有料记忆
OUT 506.08  ; #2-1电池注氦阀开条件
LD TR0
LD 506.08  ; #2-1电池注氦阀开条件
OR 606.08  ; #2-1电池注氦阀开[A]
ANDLD
ANDNOT 823.12  ; #2-1电池注氦阀开到位标志
AND 823.09  ; #2-1电池抽真空阀关到位标志
AND 824.01  ; #2-1电池破真空阀关到位标志
ANDNOT 516.08  ; #2-1电池注氦阀关条件
OUT 606.08  ; #2-1电池注氦阀开[A]
LD TR0
LD D1096.08  ; #2腔体机构关电池注氦阀（自动步）
OR D1100.07  ; #2腔体机构关#2-1电池注氦阀（自动单检步）
ANDLD
OUT 516.08  ; #2-1电池注氦阀关条件
LD TR0
LD 516.08  ; #2-1电池注氦阀关条件
OR 616.08  ; #2-1电池注氦阀关[A]
ANDLD
ANDNOT 823.13  ; #2-1电池注氦阀关到位标志
ANDNOT 506.08  ; #2-1电池注氦阀开条件
OUT 616.08  ; #2-1电池注氦阀关[A]

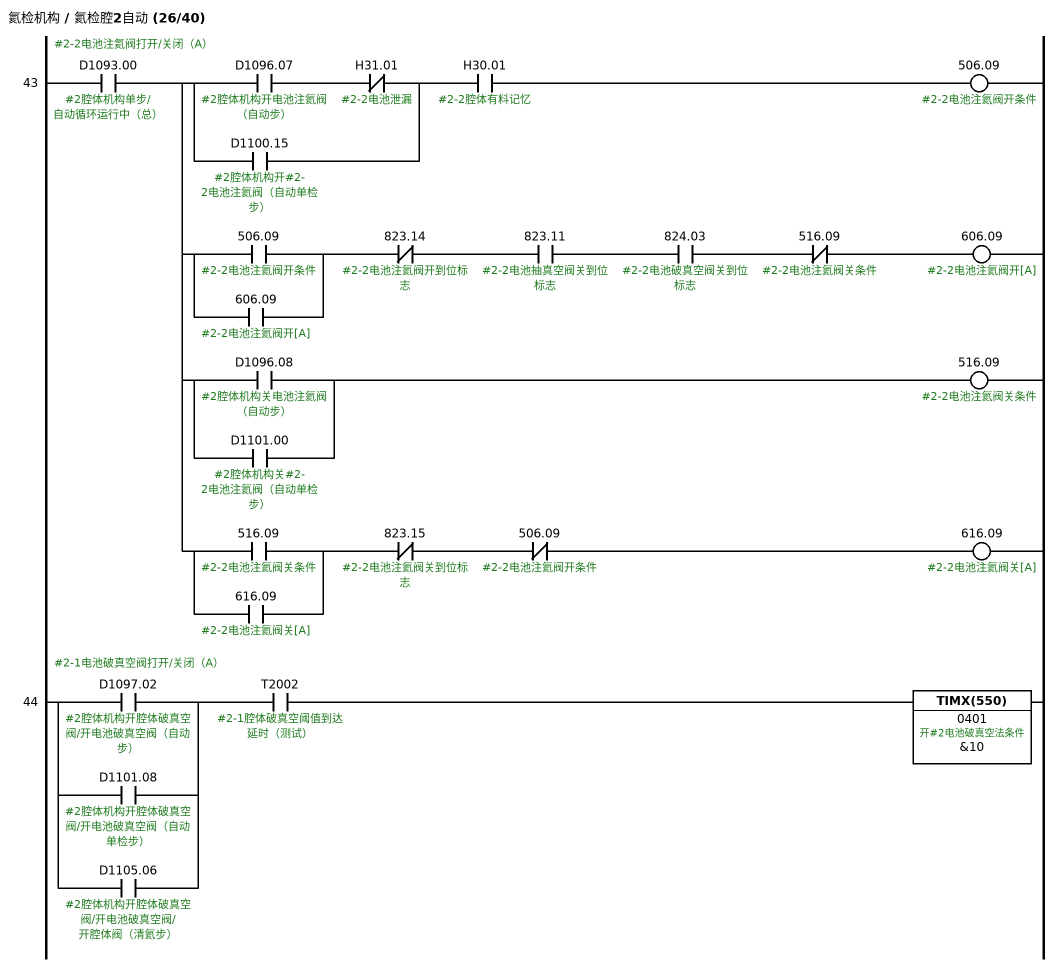
; rung 43: #2-2电池注氦阀打开/关闭（A）
LD D1093.00  ; #2腔体机构单步/自动循环运行中（总）
OUT TR0
LD D1096.07  ; #2腔体机构开电池注氦阀（自动步）
ANDNOT H31.01  ; #2-2电池泄漏
OR D1100.15  ; #2腔体机构开#2-2电池注氦阀（自动单检步）
ANDLD
AND H30.01  ; #2-2腔体有料记忆
OUT 506.09  ; #2-2电池注氦阀开条件
LD TR0
LD 506.09  ; #2-2电池注氦阀开条件
OR 606.09  ; #2-2电池注氦阀开[A]
ANDLD
ANDNOT 823.14  ; #2-2电池注氦阀开到位标志
AND 823.11  ; #2-2电池抽真空阀关到位标志
AND 824.03  ; #2-2电池破真空阀关到位标志
ANDNOT 516.09  ; #2-2电池注氦阀关条件
OUT 606.09  ; #2-2电池注氦阀开[A]
LD TR0
LD D1096.08  ; #2腔体机构关电池注氦阀（自动步）
OR D1101.00  ; #2腔体机构关#2-2电池注氦阀（自动单检步）
ANDLD
OUT 516.09  ; #2-2电池注氦阀关条件
LD TR0
LD 516.09  ; #2-2电池注氦阀关条件
OR 616.09  ; #2-2电池注氦阀关[A]
ANDLD
ANDNOT 823.15  ; #2-2电池注氦阀关到位标志
ANDNOT 506.09  ; #2-2电池注氦阀开条件
OUT 616.09  ; #2-2电池注氦阀关[A]
; rung 44: #2-1电池破真空阀打开/关闭（A）
LD D1097.02  ; #2腔体机构开腔体破真空阀/开电池破真空阀（自动步）
OR D1101.08  ; #2腔体机构开腔体破真空阀/开电池破真空阀（自动单检步）
OR D1105.06  ; #2腔体机构开腔体破真空阀/开电池破真空阀/开腔体阀（清氦步）
AND T2002  ; #2-1腔体破真空阈值到达延时（测试）
TIMX(550) 0401 &10  ; 开#2电池破真空法条件

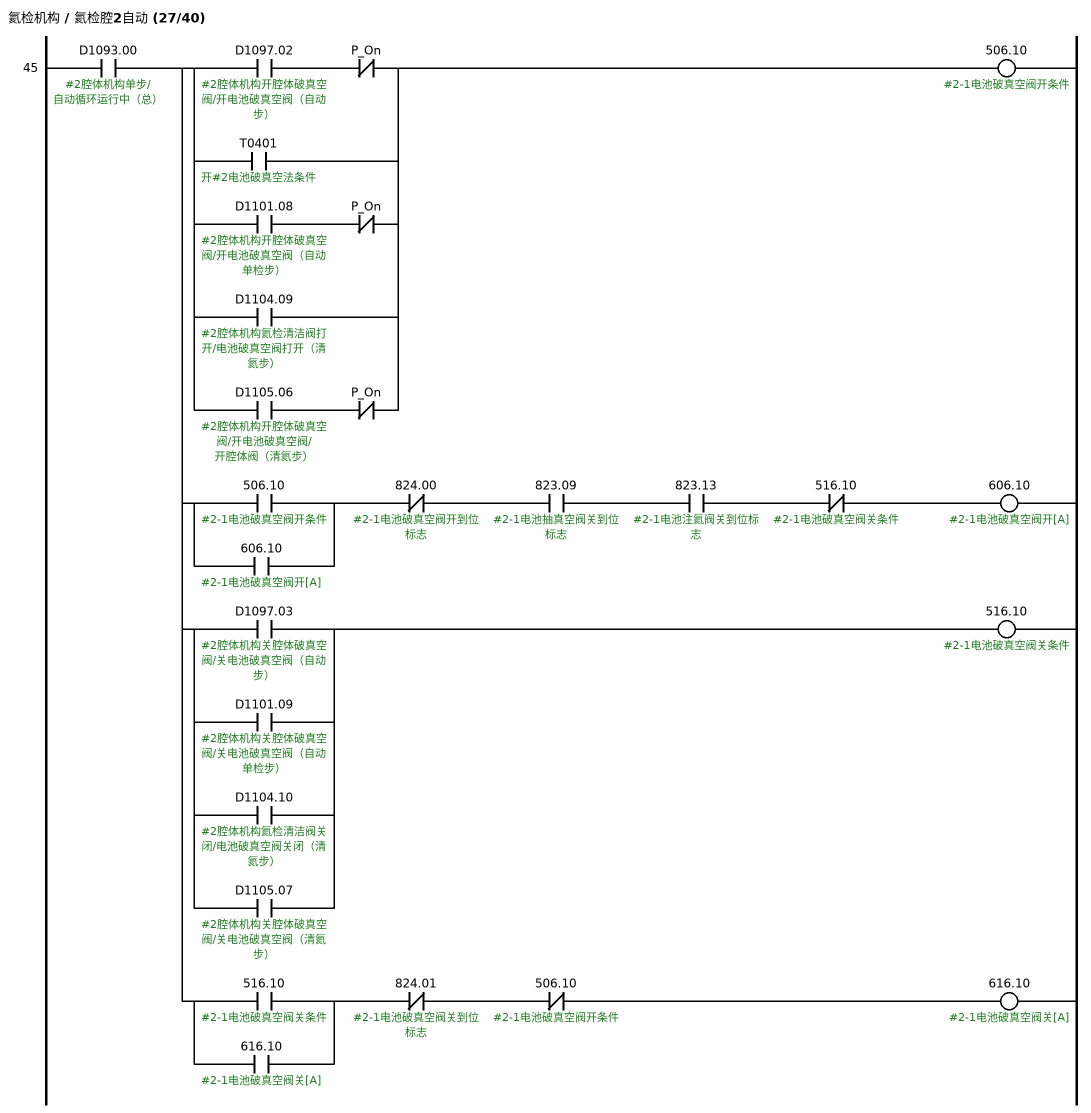
; rung 45
LD D1093.00  ; #2腔体机构单步/自动循环运行中（总）
OUT TR0
LD D1097.02  ; #2腔体机构开腔体破真空阀/开电池破真空阀（自动步）
ANDNOT P_On
OR T0401  ; 开#2电池破真空法条件
LD D1101.08  ; #2腔体机构开腔体破真空阀/开电池破真空阀（自动单检步）
ANDNOT P_On
ORLD
OR D1104.09  ; #2腔体机构氦检清洁阀打开/电池破真空阀打开（清氦步）
LD D1105.06  ; #2腔体机构开腔体破真空阀/开电池破真空阀/开腔体阀（清氦步）
ANDNOT P_On
ORLD
ANDLD
OUT 506.10  ; #2-1电池破真空阀开条件
LD TR0
LD 506.10  ; #2-1电池破真空阀开条件
OR 606.10  ; #2-1电池破真空阀开[A]
ANDLD
ANDNOT 824.00  ; #2-1电池破真空阀开到位标志
AND 823.09  ; #2-1电池抽真空阀关到位标志
AND 823.13  ; #2-1电池注氦阀关到位标志
ANDNOT 516.10  ; #2-1电池破真空阀关条件
OUT 606.10  ; #2-1电池破真空阀开[A]
LD TR0
LD D1097.03  ; #2腔体机构关腔体破真空阀/关电池破真空阀（自动步）
OR D1101.09  ; #2腔体机构关腔体破真空阀/关电池破真空阀（自动单检步）
OR D1104.10  ; #2腔体机构氦检清洁阀关闭/电池破真空阀关闭（清氦步）
OR D1105.07  ; #2腔体机构关腔体破真空阀/关电池破真空阀（清氦步）
ANDLD
OUT 516.10  ; #2-1电池破真空阀关条件
LD TR0
LD 516.10  ; #2-1电池破真空阀关条件
OR 616.10  ; #2-1电池破真空阀关[A]
ANDLD
ANDNOT 824.01  ; #2-1电池破真空阀关到位标志
ANDNOT 506.10  ; #2-1电池破真空阀开条件
OUT 616.10  ; #2-1电池破真空阀关[A]

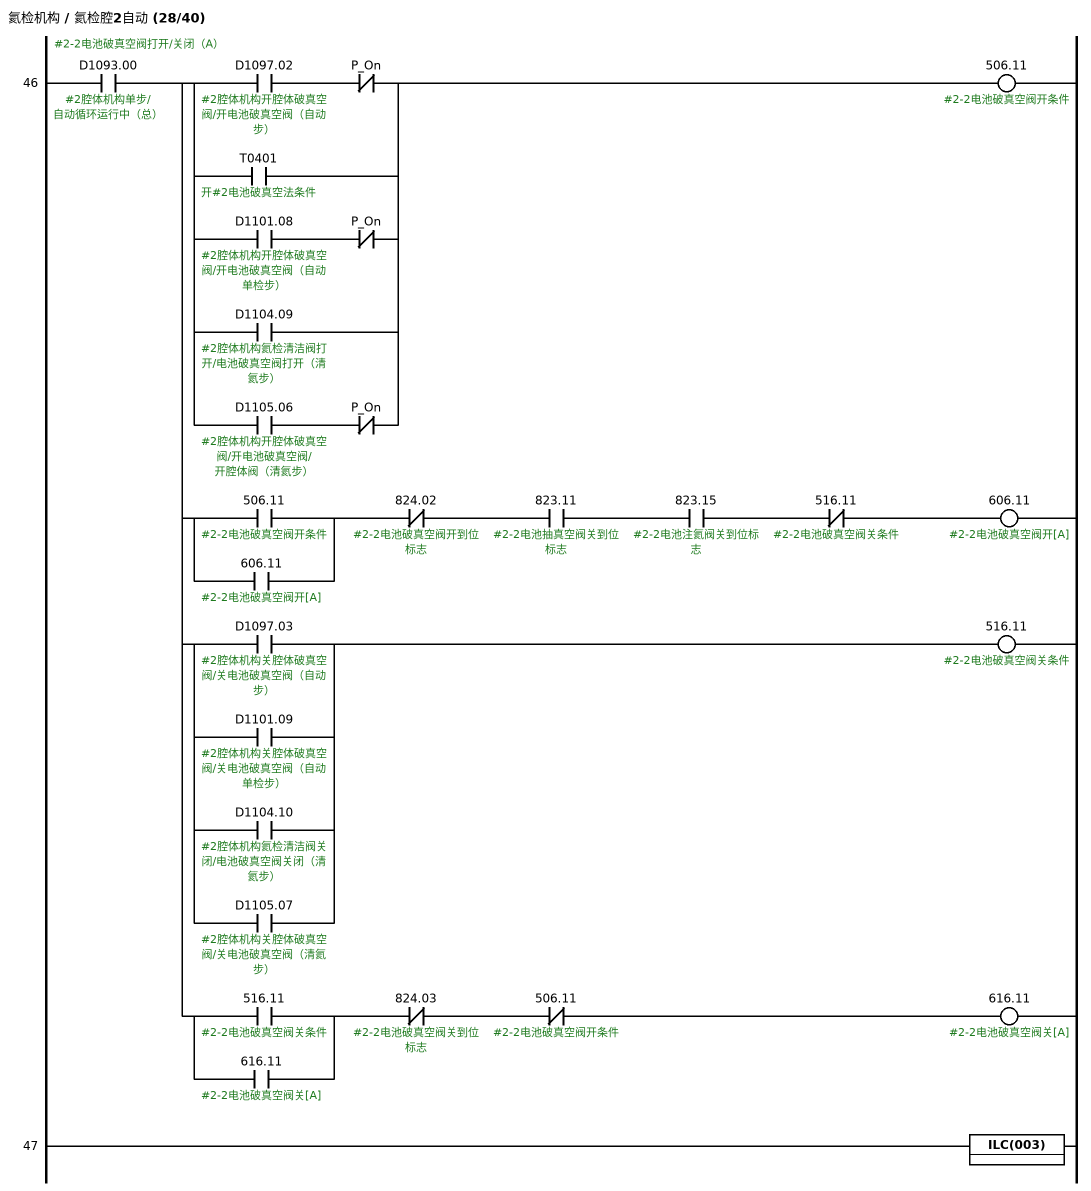
; rung 46: #2-2电池破真空阀打开/关闭（A）
LD D1093.00  ; #2腔体机构单步/自动循环运行中（总）
OUT TR0
LD D1097.02  ; #2腔体机构开腔体破真空阀/开电池破真空阀（自动步）
ANDNOT P_On
OR T0401  ; 开#2电池破真空法条件
LD D1101.08  ; #2腔体机构开腔体破真空阀/开电池破真空阀（自动单检步）
ANDNOT P_On
ORLD
OR D1104.09  ; #2腔体机构氦检清洁阀打开/电池破真空阀打开（清氦步）
LD D1105.06  ; #2腔体机构开腔体破真空阀/开电池破真空阀/开腔体阀（清氦步）
ANDNOT P_On
ORLD
ANDLD
OUT 506.11  ; #2-2电池破真空阀开条件
LD TR0
LD 506.11  ; #2-2电池破真空阀开条件
OR 606.11  ; #2-2电池破真空阀开[A]
ANDLD
ANDNOT 824.02  ; #2-2电池破真空阀开到位标志
AND 823.11  ; #2-2电池抽真空阀关到位标志
AND 823.15  ; #2-2电池注氦阀关到位标志
ANDNOT 516.11  ; #2-2电池破真空阀关条件
OUT 606.11  ; #2-2电池破真空阀开[A]
LD TR0
LD D1097.03  ; #2腔体机构关腔体破真空阀/关电池破真空阀（自动步）
OR D1101.09  ; #2腔体机构关腔体破真空阀/关电池破真空阀（自动单检步）
OR D1104.10  ; #2腔体机构氦检清洁阀关闭/电池破真空阀关闭（清氦步）
OR D1105.07  ; #2腔体机构关腔体破真空阀/关电池破真空阀（清氦步）
ANDLD
OUT 516.11  ; #2-2电池破真空阀关条件
LD TR0
LD 516.11  ; #2-2电池破真空阀关条件
OR 616.11  ; #2-2电池破真空阀关[A]
ANDLD
ANDNOT 824.03  ; #2-2电池破真空阀关到位标志
ANDNOT 506.11  ; #2-2电池破真空阀开条件
OUT 616.11  ; #2-2电池破真空阀关[A]
; rung 47
ILC(003)

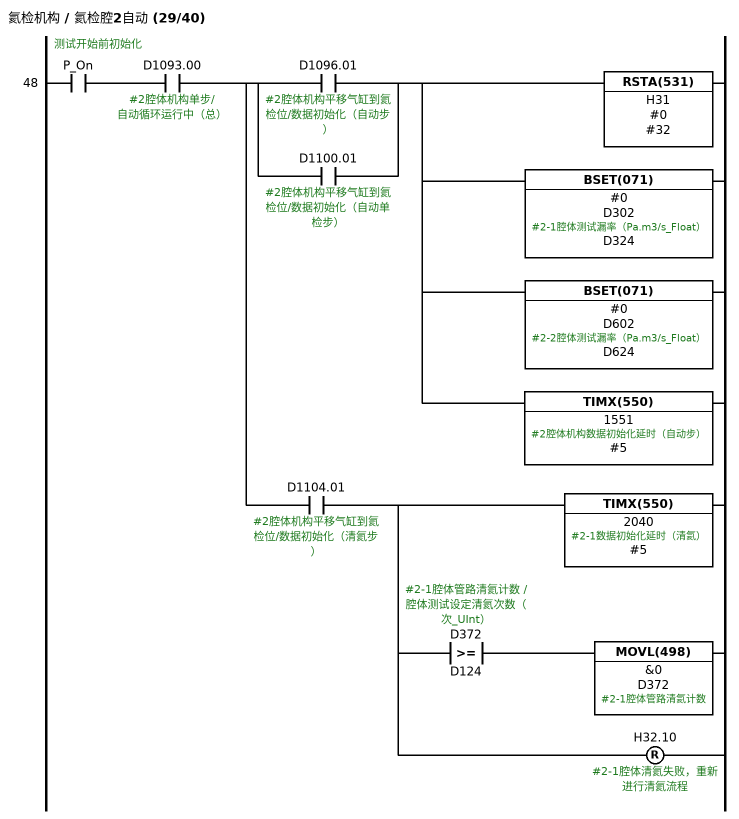
; rung 48: 测试开始前初始化
LD P_On
AND D1093.00  ; #2腔体机构单步/自动循环运行中（总）
OUT TR0
LD D1096.01  ; #2腔体机构平移气缸到氦检位/数据初始化（自动步）
OR D1100.01  ; #2腔体机构平移气缸到氦检位/数据初始化（自动单检步）
ANDLD
RSTA(531) H31 #0 #32
BSET(071) #0 D302 D324  ; #2-1腔体测试漏率（Pa.m3/s_Float）
BSET(071) #0 D602 D624  ; #2-2腔体测试漏率（Pa.m3/s_Float）
TIMX(550) 1551 #5  ; #2腔体机构数据初始化延时（自动步）
LD TR0
AND D1104.01  ; #2腔体机构平移气缸到氦检位/数据初始化（清氦步）
OUT TR0
TIMX(550) 2040 #5  ; #2-1数据初始化延时（清氦）
AND>=(325) D372 D124  ; #2-1腔体管路清氦计数, 腔体测试设定清氦次数（次_UInt）
MOVL(498) &0 D372  ; #2-1腔体管路清氦计数
LD TR0
RSET H32.10  ; #2-1腔体清氦失败，重新进行清氦流程

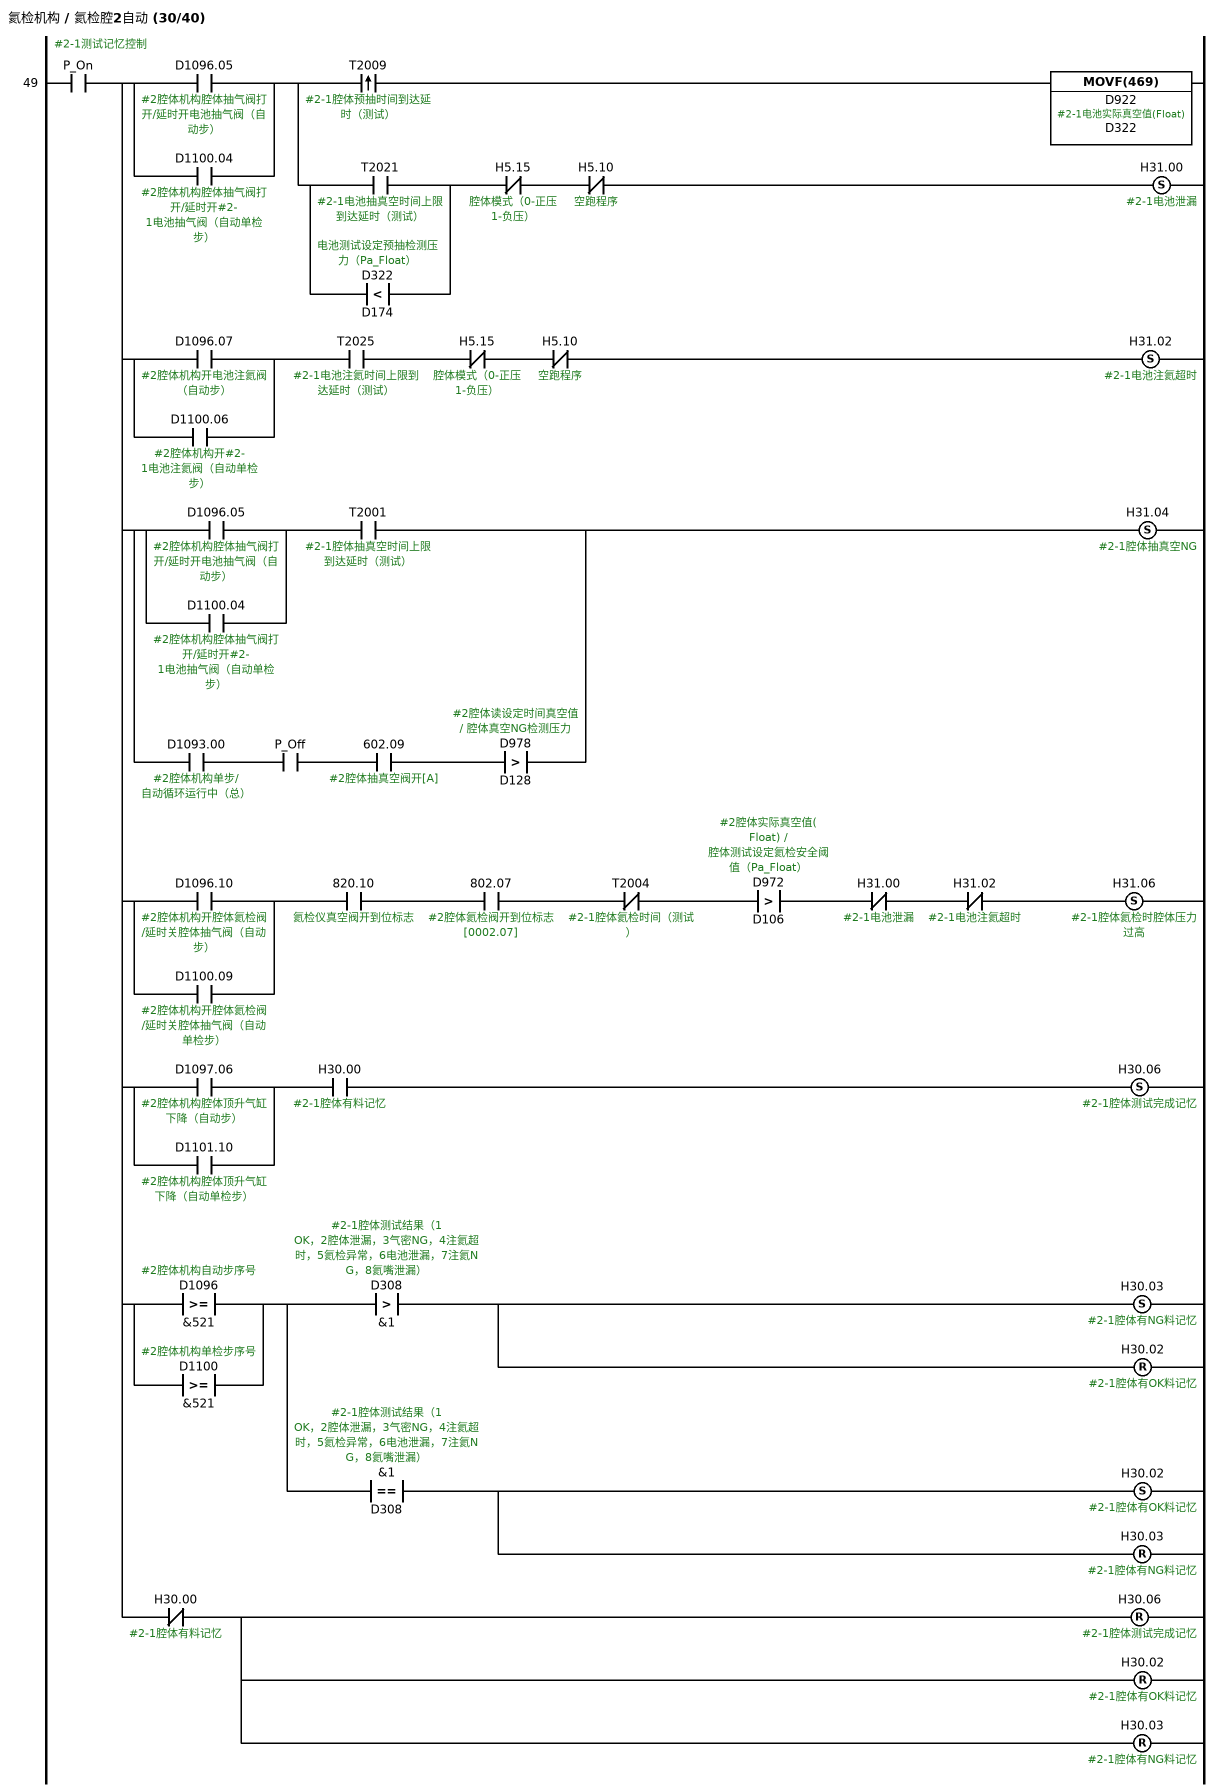
; rung 49: #2-1测试记忆控制
LD P_On
OUT TR0
LD D1096.05  ; #2腔体机构腔体抽气阀打开/延时开电池抽气阀（自动步）
OR D1100.04  ; #2腔体机构腔体抽气阀打开/延时开#2-1电池抽气阀（自动单检步）
ANDLD
OUT TR1
@AND T2009  ; #2-1腔体预抽时间到达延时（测试）
MOVF(469) D922 D322  ; #2-1电池实际真空值(Float)
LD TR1
LD T2021  ; #2-1电池抽真空时间上限到达延时（测试）
OR<F(331) D322 D174  ; 电池测试设定预抽检测压力（Pa_Float）
ANDLD
ANDNOT H5.15  ; 腔体模式（0-正压 1-负压）
ANDNOT H5.10  ; 空跑程序
SET H31.00  ; #2-1电池泄漏
LD TR0
LD D1096.07  ; #2腔体机构开电池注氦阀（自动步）
OR D1100.06  ; #2腔体机构开#2-1电池注氦阀（自动单检步）
ANDLD
AND T2025  ; #2-1电池注氦时间上限到达延时（测试）
ANDNOT H5.15  ; 腔体模式（0-正压 1-负压）
ANDNOT H5.10  ; 空跑程序
SET H31.02  ; #2-1电池注氦超时
LD TR0
LD D1096.05  ; #2腔体机构腔体抽气阀打开/延时开电池抽气阀（自动步）
OR D1100.04  ; #2腔体机构腔体抽气阀打开/延时开#2-1电池抽气阀（自动单检步）
AND T2001  ; #2-1腔体抽真空时间上限到达延时（测试）
LD D1093.00  ; #2腔体机构单步/自动循环运行中（总）
AND P_Off
AND 602.09  ; #2腔体抽真空阀开[A]
AND>F(333) D978 D128  ; #2腔体读设定时间真空值, 腔体真空NG检测压力
ORLD
ANDLD
SET H31.04  ; #2-1腔体抽真空NG
LD TR0
LD D1096.10  ; #2腔体机构开腔体氦检阀/延时关腔体抽气阀（自动步）
OR D1100.09  ; #2腔体机构开腔体氦检阀/延时关腔体抽气阀（自动单检步）
ANDLD
AND 820.10  ; 氦检仪真空阀开到位标志
AND 802.07  ; #2腔体氦检阀开到位标志[0002.07]
ANDNOT T2004  ; #2-1腔体氦检时间（测试）
AND>F(333) D972 D106  ; #2腔体实际真空值(Float), 腔体测试设定氦检安全阈值（Pa_Float）
ANDNOT H31.00  ; #2-1电池泄漏
ANDNOT H31.02  ; #2-1电池注氦超时
SET H31.06  ; #2-1腔体氦检时腔体压力过高
LD TR0
LD D1097.06  ; #2腔体机构腔体顶升气缸下降（自动步）
OR D1101.10  ; #2腔体机构腔体顶升气缸下降（自动单检步）
ANDLD
AND H30.00  ; #2-1腔体有料记忆
SET H30.06  ; #2-1腔体测试完成记忆
LD TR0
LD>=L(326) D1096 &521  ; #2腔体机构自动步序号
OR>=L(326) D1100 &521  ; #2腔体机构单检步序号
ANDLD
OUT TR1
AND>(320) D308 &1  ; #2-1腔体测试结果（1 OK，2腔体泄漏，3气密NG，4注氦超时，5氦检异常，6电池泄漏，7注氦NG，8氦嘴泄漏）
SET H30.03  ; #2-1腔体有NG料记忆
RSET H30.02  ; #2-1腔体有OK料记忆
LD TR1
AND=(300) &1 D308  ; #2-1腔体测试结果（1 OK，2腔体泄漏，3气密NG，4注氦超时，5氦检异常，6电池泄漏，7注氦NG，8氦嘴泄漏）
SET H30.02  ; #2-1腔体有OK料记忆
RSET H30.03  ; #2-1腔体有NG料记忆
LD TR0
ANDNOT H30.00  ; #2-1腔体有料记忆
RSET H30.06  ; #2-1腔体测试完成记忆
RSET H30.02  ; #2-1腔体有OK料记忆
RSET H30.03  ; #2-1腔体有NG料记忆

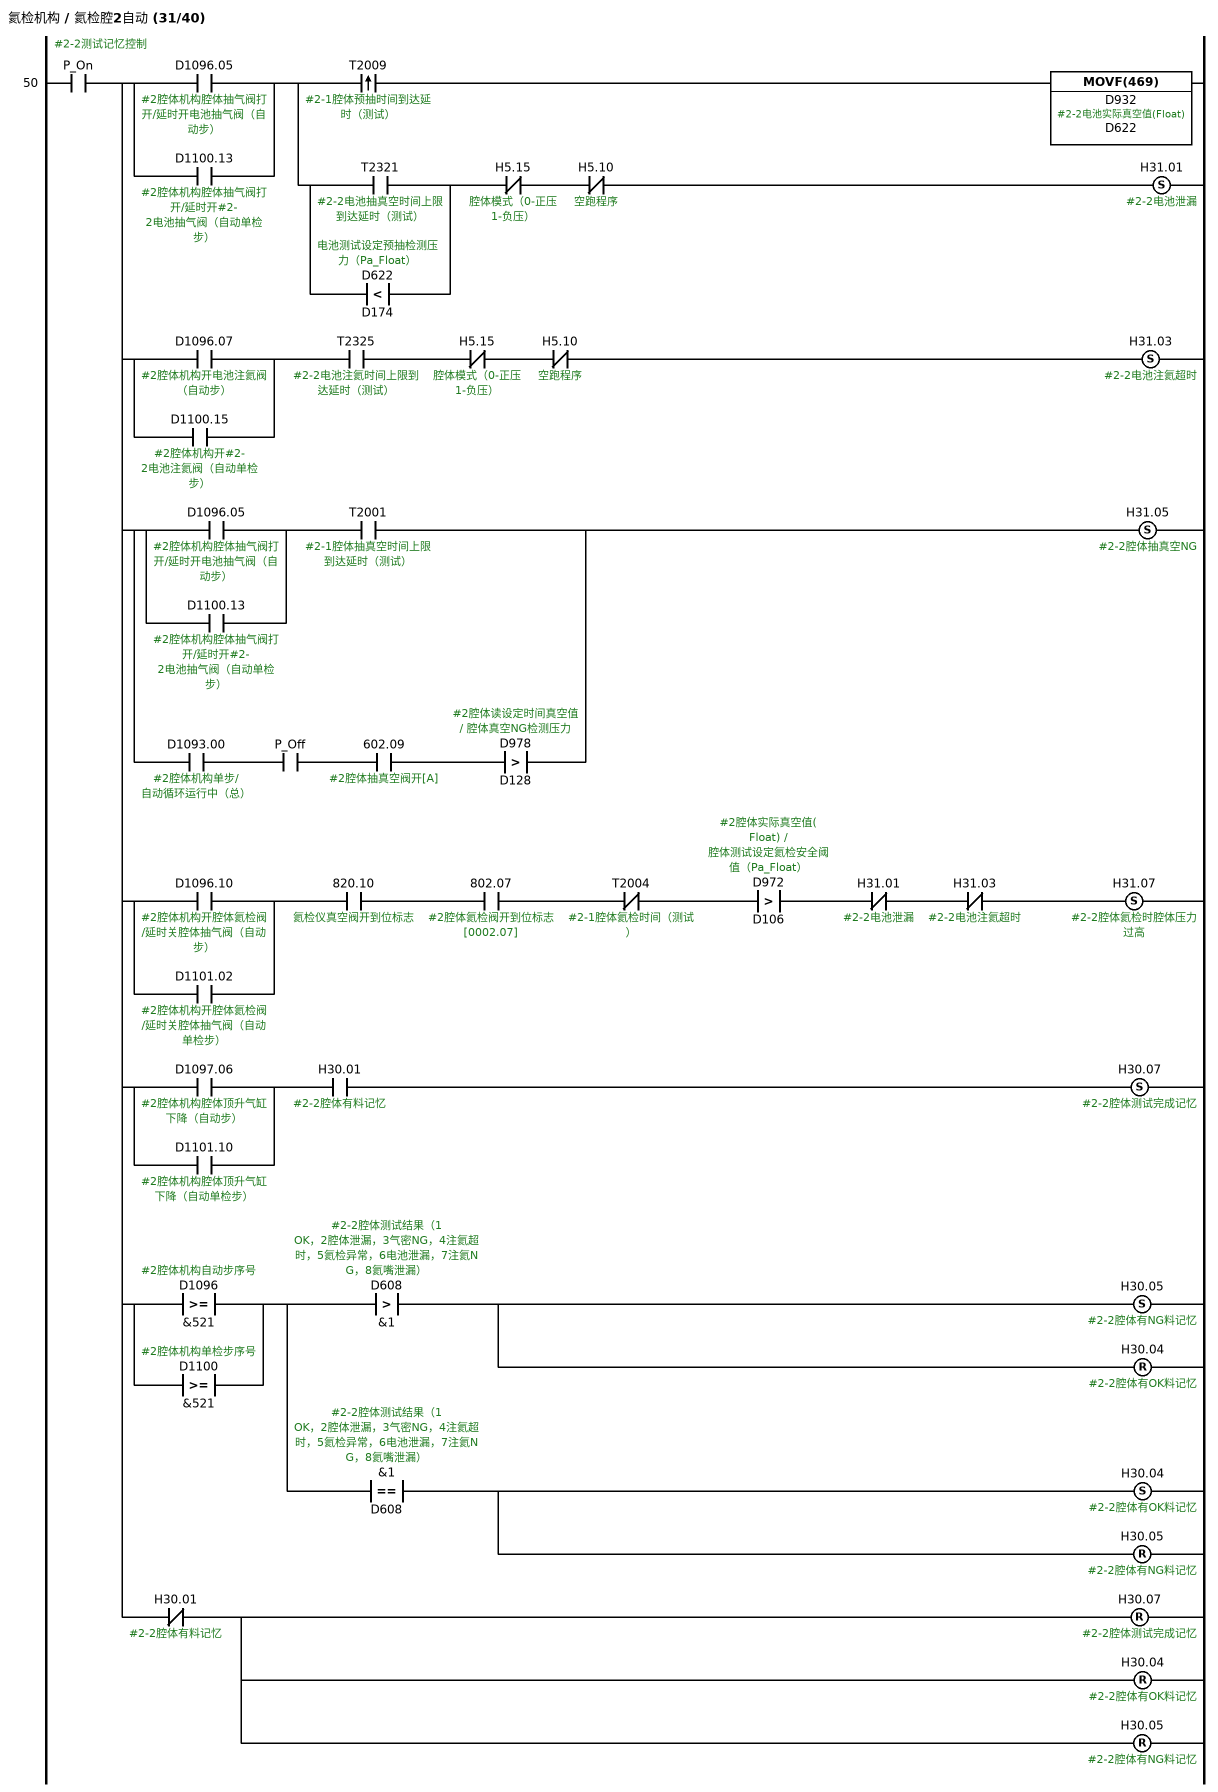
; rung 50: #2-2测试记忆控制
LD P_On
OUT TR0
LD D1096.05  ; #2腔体机构腔体抽气阀打开/延时开电池抽气阀（自动步）
OR D1100.13  ; #2腔体机构腔体抽气阀打开/延时开#2-2电池抽气阀（自动单检步）
ANDLD
OUT TR1
@AND T2009  ; #2-1腔体预抽时间到达延时（测试）
MOVF(469) D932 D622  ; #2-2电池实际真空值(Float)
LD TR1
LD T2321  ; #2-2电池抽真空时间上限到达延时（测试）
OR<F(331) D622 D174  ; 电池测试设定预抽检测压力（Pa_Float）
ANDLD
ANDNOT H5.15  ; 腔体模式（0-正压 1-负压）
ANDNOT H5.10  ; 空跑程序
SET H31.01  ; #2-2电池泄漏
LD TR0
LD D1096.07  ; #2腔体机构开电池注氦阀（自动步）
OR D1100.15  ; #2腔体机构开#2-2电池注氦阀（自动单检步）
ANDLD
AND T2325  ; #2-2电池注氦时间上限到达延时（测试）
ANDNOT H5.15  ; 腔体模式（0-正压 1-负压）
ANDNOT H5.10  ; 空跑程序
SET H31.03  ; #2-2电池注氦超时
LD TR0
LD D1096.05  ; #2腔体机构腔体抽气阀打开/延时开电池抽气阀（自动步）
OR D1100.13  ; #2腔体机构腔体抽气阀打开/延时开#2-2电池抽气阀（自动单检步）
AND T2001  ; #2-1腔体抽真空时间上限到达延时（测试）
LD D1093.00  ; #2腔体机构单步/自动循环运行中（总）
AND P_Off
AND 602.09  ; #2腔体抽真空阀开[A]
AND>F(333) D978 D128  ; #2腔体读设定时间真空值, 腔体真空NG检测压力
ORLD
ANDLD
SET H31.05  ; #2-2腔体抽真空NG
LD TR0
LD D1096.10  ; #2腔体机构开腔体氦检阀/延时关腔体抽气阀（自动步）
OR D1101.02  ; #2腔体机构开腔体氦检阀/延时关腔体抽气阀（自动单检步）
ANDLD
AND 820.10  ; 氦检仪真空阀开到位标志
AND 802.07  ; #2腔体氦检阀开到位标志[0002.07]
ANDNOT T2004  ; #2-1腔体氦检时间（测试）
AND>F(333) D972 D106  ; #2腔体实际真空值(Float), 腔体测试设定氦检安全阈值（Pa_Float）
ANDNOT H31.01  ; #2-2电池泄漏
ANDNOT H31.03  ; #2-2电池注氦超时
SET H31.07  ; #2-2腔体氦检时腔体压力过高
LD TR0
LD D1097.06  ; #2腔体机构腔体顶升气缸下降（自动步）
OR D1101.10  ; #2腔体机构腔体顶升气缸下降（自动单检步）
ANDLD
AND H30.01  ; #2-2腔体有料记忆
SET H30.07  ; #2-2腔体测试完成记忆
LD TR0
LD>=L(326) D1096 &521  ; #2腔体机构自动步序号
OR>=L(326) D1100 &521  ; #2腔体机构单检步序号
ANDLD
OUT TR1
AND>(320) D608 &1  ; #2-2腔体测试结果（1 OK，2腔体泄漏，3气密NG，4注氦超时，5氦检异常，6电池泄漏，7注氦NG，8氦嘴泄漏）
SET H30.05  ; #2-2腔体有NG料记忆
RSET H30.04  ; #2-2腔体有OK料记忆
LD TR1
AND=(300) &1 D608  ; #2-2腔体测试结果（1 OK，2腔体泄漏，3气密NG，4注氦超时，5氦检异常，6电池泄漏，7注氦NG，8氦嘴泄漏）
SET H30.04  ; #2-2腔体有OK料记忆
RSET H30.05  ; #2-2腔体有NG料记忆
LD TR0
ANDNOT H30.01  ; #2-2腔体有料记忆
RSET H30.07  ; #2-2腔体测试完成记忆
RSET H30.04  ; #2-2腔体有OK料记忆
RSET H30.05  ; #2-2腔体有NG料记忆

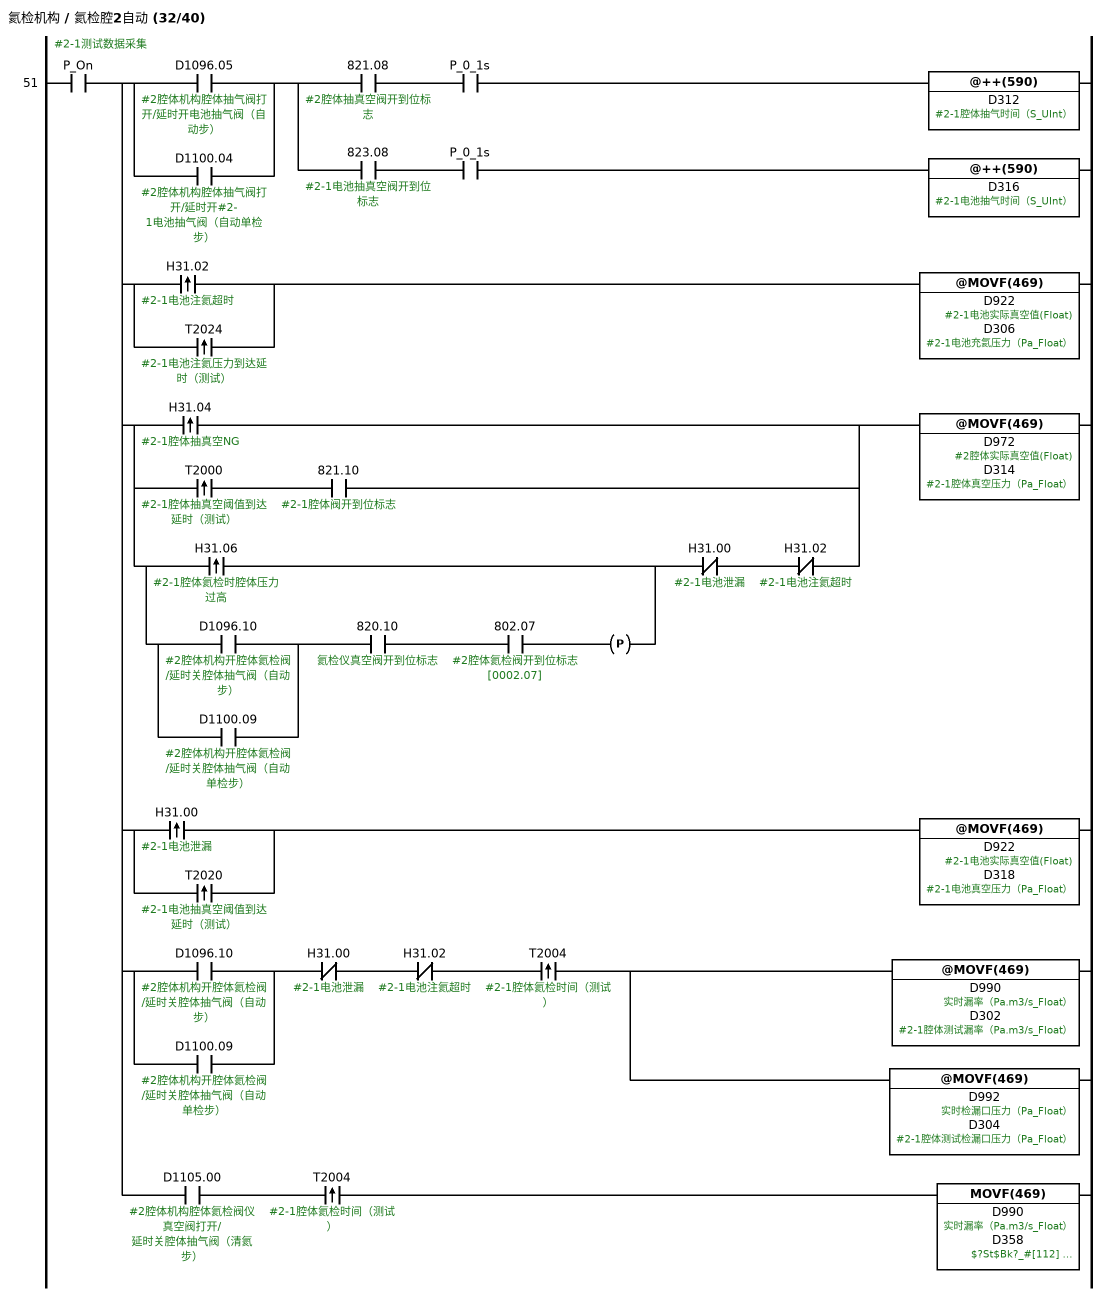
; rung 51: #2-1测试数据采集
LD P_On
OUT TR0
LD D1096.05  ; #2腔体机构腔体抽气阀打开/延时开电池抽气阀（自动步）
OR D1100.04  ; #2腔体机构腔体抽气阀打开/延时开#2-1电池抽气阀（自动单检步）
ANDLD
OUT TR1
AND 821.08  ; #2腔体抽真空阀开到位标志
AND P_0_1s
@++(590) D312  ; #2-1腔体抽气时间（S_UInt）
LD TR1
AND 823.08  ; #2-1电池抽真空阀开到位标志
AND P_0_1s
@++(590) D316  ; #2-1电池抽气时间（S_UInt）
LD TR0
@LD H31.02  ; #2-1电池注氦超时
@OR T2024  ; #2-1电池注氦压力到达延时（测试）
ANDLD
@MOVF(469) D922 D306  ; #2-1电池实际真空值(Float), #2-1电池充氦压力（Pa_Float）
LD TR0
@LD H31.04  ; #2-1腔体抽真空NG
@LD T2000  ; #2-1腔体抽真空阈值到达延时（测试）
AND 821.10  ; #2-1腔体阀开到位标志
ORLD
@LD H31.06  ; #2-1腔体氦检时腔体压力过高
LD D1096.10  ; #2腔体机构开腔体氦检阀/延时关腔体抽气阀（自动步）
OR D1100.09  ; #2腔体机构开腔体氦检阀/延时关腔体抽气阀（自动单检步）
AND 820.10  ; 氦检仪真空阀开到位标志
AND 802.07  ; #2腔体氦检阀开到位标志[0002.07]
UP(521)
ORLD
ANDNOT H31.00  ; #2-1电池泄漏
ANDNOT H31.02  ; #2-1电池注氦超时
ORLD
ANDLD
@MOVF(469) D972 D314  ; #2腔体实际真空值(Float), #2-1腔体真空压力（Pa_Float）
LD TR0
@LD H31.00  ; #2-1电池泄漏
@OR T2020  ; #2-1电池抽真空阈值到达延时（测试）
ANDLD
@MOVF(469) D922 D318  ; #2-1电池实际真空值(Float), #2-1电池真空压力（Pa_Float）
LD TR0
LD D1096.10  ; #2腔体机构开腔体氦检阀/延时关腔体抽气阀（自动步）
OR D1100.09  ; #2腔体机构开腔体氦检阀/延时关腔体抽气阀（自动单检步）
ANDLD
ANDNOT H31.00  ; #2-1电池泄漏
ANDNOT H31.02  ; #2-1电池注氦超时
@AND T2004  ; #2-1腔体氦检时间（测试）
@MOVF(469) D990 D302  ; 实时漏率（Pa.m3/s_Float）, #2-1腔体测试漏率（Pa.m3/s_Float）
@MOVF(469) D992 D304  ; 实时检漏口压力（Pa_Float）, #2-1腔体测试检漏口压力（Pa_Float）
LD TR0
AND D1105.00  ; #2腔体机构腔体氦检阀仪真空阀打开/延时关腔体抽气阀（清氦步）
@AND T2004  ; #2-1腔体氦检时间（测试）
MOVF(469) D990 D358  ; 实时漏率（Pa.m3/s_Float）, $?St$Bk?_#[112] / #2-1清氦泄漏率（清氦） / $?St$Bk?_#[112]

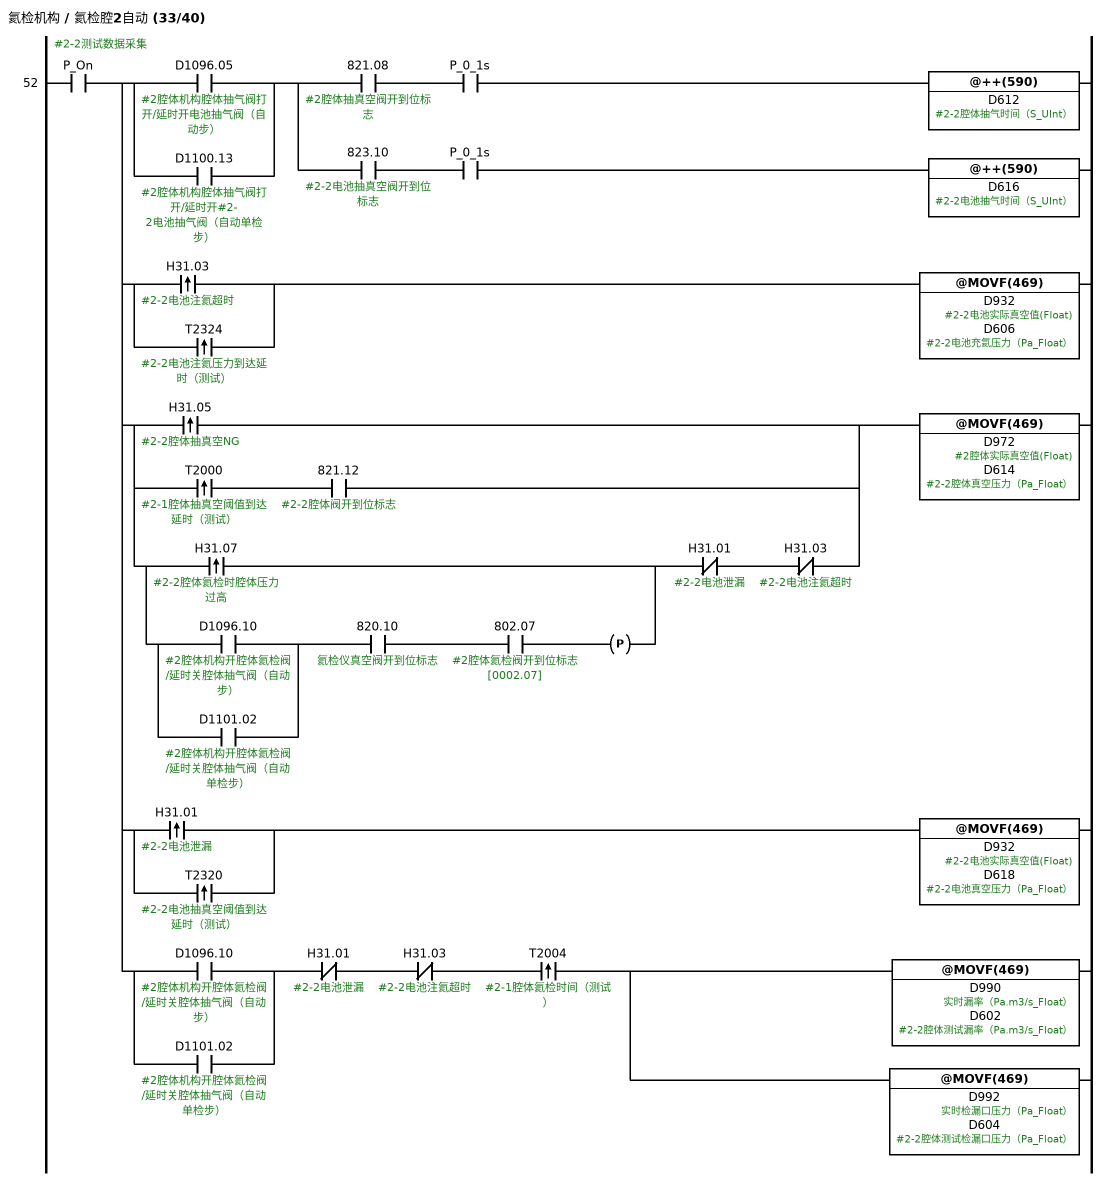
; rung 52: #2-2测试数据采集
LD P_On
OUT TR0
LD D1096.05  ; #2腔体机构腔体抽气阀打开/延时开电池抽气阀（自动步）
OR D1100.13  ; #2腔体机构腔体抽气阀打开/延时开#2-2电池抽气阀（自动单检步）
ANDLD
OUT TR1
AND 821.08  ; #2腔体抽真空阀开到位标志
AND P_0_1s
@++(590) D612  ; #2-2腔体抽气时间（S_UInt）
LD TR1
AND 823.10  ; #2-2电池抽真空阀开到位标志
AND P_0_1s
@++(590) D616  ; #2-2电池抽气时间（S_UInt）
LD TR0
@LD H31.03  ; #2-2电池注氦超时
@OR T2324  ; #2-2电池注氦压力到达延时（测试）
ANDLD
@MOVF(469) D932 D606  ; #2-2电池实际真空值(Float), #2-2电池充氦压力（Pa_Float）
LD TR0
@LD H31.05  ; #2-2腔体抽真空NG
@LD T2000  ; #2-1腔体抽真空阈值到达延时（测试）
AND 821.12  ; #2-2腔体阀开到位标志
ORLD
@LD H31.07  ; #2-2腔体氦检时腔体压力过高
LD D1096.10  ; #2腔体机构开腔体氦检阀/延时关腔体抽气阀（自动步）
OR D1101.02  ; #2腔体机构开腔体氦检阀/延时关腔体抽气阀（自动单检步）
AND 820.10  ; 氦检仪真空阀开到位标志
AND 802.07  ; #2腔体氦检阀开到位标志[0002.07]
UP(521)
ORLD
ANDNOT H31.01  ; #2-2电池泄漏
ANDNOT H31.03  ; #2-2电池注氦超时
ORLD
ANDLD
@MOVF(469) D972 D614  ; #2腔体实际真空值(Float), #2-2腔体真空压力（Pa_Float）
LD TR0
@LD H31.01  ; #2-2电池泄漏
@OR T2320  ; #2-2电池抽真空阈值到达延时（测试）
ANDLD
@MOVF(469) D932 D618  ; #2-2电池实际真空值(Float), #2-2电池真空压力（Pa_Float）
LD TR0
LD D1096.10  ; #2腔体机构开腔体氦检阀/延时关腔体抽气阀（自动步）
OR D1101.02  ; #2腔体机构开腔体氦检阀/延时关腔体抽气阀（自动单检步）
ANDLD
ANDNOT H31.01  ; #2-2电池泄漏
ANDNOT H31.03  ; #2-2电池注氦超时
@AND T2004  ; #2-1腔体氦检时间（测试）
@MOVF(469) D990 D602  ; 实时漏率（Pa.m3/s_Float）, #2-2腔体测试漏率（Pa.m3/s_Float）
@MOVF(469) D992 D604  ; 实时检漏口压力（Pa_Float）, #2-2腔体测试检漏口压力（Pa_Float）

